LIN {X 0,Y 168.921,Z 1046.444,A -85,B 0,C 180,E1 28928.904,E2 28928.904} C_VEL
LIN {X 0,Y 193.808,Z 1028.505,A -85,B 0,C 180,E1 28941.439,E2 28941.439} C_VEL
LIN {X 0,Y 223.999,Z 1004.253,A -85,B 0,C 180,E1 28950.581,E2 28950.581} C_VEL
LIN {X 0,Y 255.108,Z 974.593,A -85,B 0,C 180,E1 28956.989,E2 28956.989} C_VEL
LIN {X 0,Y 284.282,Z 940.686,A -85,B 0,C 180,E1 28961.432,E2 28961.432} C_VEL
LIN {X 0,Y 287.15,Z 937.068,A -85,B 0,C 180,E1 28961.796,E2 28961.796} C_VEL
LIN {X 0,Y 289.842,Z 928.042,A -85,B 0,C 180,E1 28965.797,E2 28965.797} C_VEL
LIN {X 0,Y 291.827,Z 919.586,A -85,B 0,C 180,E1 28971.585,E2 28971.585} C_VEL
LIN {X 0,Y 293.357,Z 915.265,A -85,B 0,C 180,E1 28977.034,E2 28977.034} C_VEL
LIN {X 0,Y 293.788,Z 914.928,A -85,B 0,C 180,E1 28979.995,E2 28979.995} C_VEL
LIN {X 0,Y 292.859,Z 920.588,A -85,B 0,C 180,E1 28986.732,E2 28986.732} C_VEL
LIN {X 0,Y 291.654,Z 929.151,A -85,B 0,C 180,E1 28991.99,E2 28991.99} C_VEL
LIN {X 0,Y 290.091,Z 935.801,A -85,B 0,C 180,E1 28994.874,E2 28994.874} C_VEL
LIN {X 0,Y 261.778,Z 970.623,A -85,B 0,C 180,E1 28998.746,E2 28998.746} C_VEL
LIN {X 0,Y 232.501,Z 1000.468,A -85,B 0,C 180,E1 29004.144,E2 29004.144} C_VEL
LIN {X 0,Y 202.253,Z 1026.572,A -85,B 0,C 180,E1 29012.088,E2 29012.088} C_VEL
LIN {X 0,Y 173.882,Z 1048.21,A -85,B 0,C 180,E1 29024.19,E2 29024.19} C_VEL
LIN {X 0,Y 156.367,Z 1061.241,A -85,B 0,C 180,E1 29037.787,E2 29037.787} C_VEL
LIN {X 0,Y 148.038,Z 1068.795,A -85,B 0,C 180,E1 29052.113,E2 29052.113} C_VEL
LIN {X 0,Y 145.937,Z 1071.767,A -85,B 0,C 180,E1 29064.037,E2 29064.037} C_VEL
LIN {X 0,Y 146.316,Z 1072.302,A -85,B 0,C 180,E1 29069.997,E2 29069.997} C_VEL
LIN {X 0,Y 146.516,Z 1071.402,A -85,B 0,C 180,E1 29081.935,E2 29081.935} C_VEL
LIN {X 0,Y 151.978,Z 1066.921,A -85,B 0,C 180,E1 29096.206,E2 29096.206} C_VEL
LIN {X 0,Y 168.648,Z 1055.739,A -85,B 0,C 180,E1 29112.367,E2 29112.367} C_VEL
LIN {X 0,Y 194.431,Z 1038.433,A -85,B 0,C 180,E1 29124.918,E2 29124.918} C_VEL
LIN {X 0,Y 224.573,Z 1015.903,A -85,B 0,C 180,E1 29133.68,E2 29133.68} C_VEL
LIN {X 0,Y 256.304,Z 987.953,A -85,B 0,C 180,E1 29139.894,E2 29139.894} C_VEL
LIN {X 0,Y 288.623,Z 953.147,A -85,B 0,C 180,E1 29144.481,E2 29144.481} C_VEL
LIN {X 0,Y 296.037,Z 943.922,A -85,B 0,C 180,E1 29145.338,E2 29145.338} C_VEL
LIN {X 0,Y 297.368,Z 940.896,A -85,B 0,C 180,E1 29146.446,E2 29146.446} C_VEL
LIN {X 0,Y 299.07,Z 931.533,A -85,B 0,C 180,E1 29152.728,E2 29152.728} C_VEL
LIN {X 0,Y 299.728,Z 928.149,A -85,B 0,C 180,E1 29157.107,E2 29157.107} C_VEL
LIN {X 0,Y 299.819,Z 927.494,A -85,B 0,C 180,E1 29160.005,E2 29160.005} C_VEL
LIN {X 0,Y 297.474,Z 933.11,A -85,B 0,C 180,E1 29167.322,E2 29167.322} C_VEL
LIN {X 0,Y 294.947,Z 941.251,A -85,B 0,C 180,E1 29172.533,E2 29172.533} C_VEL
LIN {X 0,Y 293.335,Z 944.677,A -85,B 0,C 180,E1 29173.859,E2 29173.859} C_VEL
LIN {X 0,Y 263.75,Z 977.365,A -85,B 0,C 180,E1 29177.989,E2 29177.989} C_VEL
LIN {X 0,Y 233.929,Z 1004.507,A -85,B 0,C 180,E1 29183.498,E2 29183.498} C_VEL
LIN {X 0,Y 204.082,Z 1027.314,A -85,B 0,C 180,E1 29191.326,E2 29191.326} C_VEL
LIN {X 0,Y 176.268,Z 1045.628,A -85,B 0,C 180,E1 29202.828,E2 29202.828} C_VEL
LIN {X 0,Y 156.666,Z 1057.623,A -85,B 0,C 180,E1 29217.862,E2 29217.862} C_VEL
LIN {X 0,Y 148.093,Z 1063.059,A -85,B 0,C 180,E1 29232.125,E2 29232.125} C_VEL
LIN {X 0,Y 146.279,Z 1064.375,A -85,B 0,C 180,E1 29250.003,E2 29250.003} C_VEL
LIN {X 0,Y 147.555,Z 1062.344,A -85,B 0,C 180,E1 29261.856,E2 29261.856} C_VEL
LIN {X 0,Y 152.427,Z 1058.204,A -85,B 0,C 180,E1 29272.752,E2 29272.752} C_VEL
LIN {X 0,Y 153.265,Z 1055.117,A -85,B 0,C 180,E1 29279.211,E2 29279.211} C_VEL
LIN {X 0,Y 155.695,Z 1051.318,A -85,B 0,C 180,E1 29285.522,E2 29285.522} C_VEL
LIN {X 0,Y 179.336,Z 1035.523,A -85,B 0,C 180,E1 29299.512,E2 29299.512} C_VEL
LIN {X 0,Y 210.143,Z 1012.776,A -85,B 0,C 180,E1 29309.927,E2 29309.927} C_VEL
LIN {X 0,Y 242.764,Z 984.247,A -85,B 0,C 180,E1 29317.038,E2 29317.038} C_VEL
LIN {X 0,Y 274.308,Z 950.43,A -85,B 0,C 180,E1 29321.97,E2 29321.97} C_VEL
LIN {X 0,Y 282.718,Z 939.972,A -85,B 0,C 180,E1 29323.075,E2 29323.075} C_VEL
LIN {X 0,Y 285.788,Z 929.836,A -85,B 0,C 180,E1 29328.525,E2 29328.525} C_VEL
LIN {X 0,Y 287.675,Z 923.701,A -85,B 0,C 180,E1 29333.947,E2 29333.947} C_VEL
LIN {X 0,Y 288.554,Z 921.686,A -85,B 0,C 180,E1 29336.984,E2 29336.984} C_VEL
LIN {X 0,Y 289.013,Z 921.304,A -85,B 0,C 180,E1 29339.995,E2 29339.995} C_VEL
LIN {X 0,Y 288.103,Z 926.168,A -85,B 0,C 180,E1 29346.033,E2 29346.033} C_VEL
LIN {X 0,Y 286.388,Z 934.915,A -85,B 0,C 180,E1 29351.687,E2 29351.687} C_VEL
LIN {X 0,Y 285.234,Z 939.354,A -85,B 0,C 180,E1 29353.657,E2 29353.657} C_VEL
LIN {X 0,Y 254.602,Z 975.363,A -85,B 0,C 180,E1 29357.758,E2 29357.758} C_VEL
LIN {X 0,Y 222.094,Z 1006.526,A -85,B 0,C 180,E1 29363.799,E2 29363.799} C_VEL
LIN {X 0,Y 192.091,Z 1030.713,A -85,B 0,C 180,E1 29371.994,E2 29371.994} C_VEL
LIN {X 0,Y 166.418,Z 1049.188,A -85,B 0,C 180,E1 29383.238,E2 29383.238} C_VEL
LIN {X 0,Y 147.059,Z 1062.863,A -85,B 0,C 180,E1 29398.984,E2 29398.984} C_VEL
LIN {X 0,Y 140.394,Z 1068.559,A -85,B 0,C 180,E1 29411.103,E2 29411.103} C_VEL
LIN {X 0,Y 138.03,Z 1071.546,A -85,B 0,C 180,E1 29423.694,E2 29423.694} C_VEL
LIN {X 0,Y 138.396,Z 1072.088,A -85,B 0,C 180,E1 29429.997,E2 29429.997} C_VEL
LIN {X 0,Y 138.722,Z 1071.199,A -85,B 0,C 180,E1 29442.617,E2 29442.617} C_VEL
LIN {X 0,Y 144.75,Z 1066.727,A -85,B 0,C 180,E1 29457.623,E2 29457.623} C_VEL
LIN {X 0,Y 162.692,Z 1055.562,A -85,B 0,C 180,E1 29474.31,E2 29474.31} C_VEL
LIN {X 0,Y 189.855,Z 1038.279,A -85,B 0,C 180,E1 29486.936,E2 29486.936} C_VEL
LIN {X 0,Y 220.041,Z 1016.621,A -85,B 0,C 180,E1 29495.338,E2 29495.338} C_VEL
LIN {X 0,Y 253.534,Z 987.948,A -85,B 0,C 180,E1 29501.593,E2 29501.593} C_VEL
LIN {X 0,Y 286.881,Z 952.718,A -85,B 0,C 180,E1 29506.063,E2 29506.063} C_VEL
LIN {X 0,Y 291.416,Z 947.157,A -85,B 0,C 180,E1 29506.56,E2 29506.56} C_VEL
LIN {X 0,Y 293.48,Z 939.749,A -85,B 0,C 180,E1 29511.094,E2 29511.094} C_VEL
LIN {X 0,Y 294.665,Z 934.317,A -85,B 0,C 180,E1 29517.057,E2 29517.057} C_VEL
LIN {X 0,Y 294.769,Z 933.639,A -85,B 0,C 180,E1 29520.005,E2 29520.005} C_VEL
LIN {X 0,Y 292.789,Z 937.807,A -85,B 0,C 180,E1 29525.947,E2 29525.947} C_VEL
LIN {X 0,Y 289.965,Z 945.492,A -85,B 0,C 180,E1 29531.508,E2 29531.508} C_VEL
LIN {X 0,Y 288.508,Z 948.427,A -85,B 0,C 180,E1 29532.691,E2 29532.691} C_VEL
LIN {X 0,Y 256.762,Z 981.946,A -85,B 0,C 180,E1 29537.013,E2 29537.013} C_VEL
LIN {X 0,Y 224.354,Z 1009.714,A -85,B 0,C 180,E1 29543.035,E2 29543.035} C_VEL
LIN {X 0,Y 194.514,Z 1031.009,A -85,B 0,C 180,E1 29551.025,E2 29551.025} C_VEL
LIN {X 0,Y 168.277,Z 1047.332,A -85,B 0,C 180,E1 29562.219,E2 29562.219} C_VEL
LIN {X 0,Y 149.856,Z 1057.809,A -85,B 0,C 180,E1 29576.211,E2 29576.211} C_VEL
LIN {X 0,Y 140.48,Z 1063.256,A -85,B 0,C 180,E1 29591.121,E2 29591.121} C_VEL
LIN {X 0,Y 137.97,Z 1064.743,A -85,B 0,C 180,E1 29603.697,E2 29603.697} C_VEL
LIN {X 0,Y 138.358,Z 1064.59,A -85,B 0,C 180,E1 29610.003,E2 29610.003} C_VEL
LIN {X 0,Y 139.83,Z 1062.527,A -85,B 0,C 180,E1 29622.694,E2 29622.694} C_VEL
LIN {X 0,Y 150.114,Z 1055,A -85,B 0,C 180,E1 29640.318,E2 29640.318} C_VEL
LIN {X 0,Y 155.695,Z 1051.318,A -85,B 0,C 180,E1 29645.522,E2 29645.522} C_VEL
LIN {X 0,Y 159.585,Z 1046.926,A -85,B 0,C 180,E1 29651.527,E2 29651.527} C_VEL
LIN {X 0,Y 164.863,Z 1041.862,A -85,B 0,C 180,E1 29657.175,E2 29657.175} C_VEL
LIN {X 0,Y 194.943,Z 1021.511,A -85,B 0,C 180,E1 29668.774,E2 29668.774} C_VEL
LIN {X 0,Y 227.398,Z 995.695,A -85,B 0,C 180,E1 29676.562,E2 29676.562} C_VEL
LIN {X 0,Y 259.168,Z 965.038,A -85,B 0,C 180,E1 29681.84,E2 29681.84} C_VEL
LIN {X 0,Y 277.327,Z 944.261,A -85,B 0,C 180,E1 29684.24,E2 29684.24} C_VEL
LIN {X 0,Y 280.428,Z 936.455,A -85,B 0,C 180,E1 29688.34,E2 29688.34} C_VEL
LIN {X 0,Y 282.59,Z 930.048,A -85,B 0,C 180,E1 29693.838,E2 29693.838} C_VEL
LIN {X 0,Y 283.64,Z 928.013,A -85,B 0,C 180,E1 29696.932,E2 29696.932} C_VEL
LIN {X 0,Y 284.164,Z 927.612,A -85,B 0,C 180,E1 29699.994,E2 29699.994} C_VEL
LIN {X 0,Y 282.944,Z 932.529,A -85,B 0,C 180,E1 29706.143,E2 29706.143} C_VEL
LIN {X 0,Y 280.729,Z 942.17,A -85,B 0,C 180,E1 29712.183,E2 29712.183} C_VEL
LIN {X 0,Y 250.587,Z 976.786,A -85,B 0,C 180,E1 29716.25,E2 29716.25} C_VEL
LIN {X 0,Y 217.78,Z 1007.215,A -85,B 0,C 180,E1 29722.087,E2 29722.087} C_VEL
LIN {X 0,Y 185.18,Z 1032.411,A -85,B 0,C 180,E1 29730.763,E2 29730.763} C_VEL
LIN {X 0,Y 156.507,Z 1051.81,A -85,B 0,C 180,E1 29743.646,E2 29743.646} C_VEL
LIN {X 0,Y 137.865,Z 1064.196,A -85,B 0,C 180,E1 29760.264,E2 29760.264} C_VEL
LIN {X 0,Y 130.923,Z 1070.144,A -85,B 0,C 180,E1 29776.612,E2 29776.612} C_VEL
LIN {X 0,Y 130.474,Z 1071.873,A -85,B 0,C 180,E1 29789.997,E2 29789.997} C_VEL
LIN {X 0,Y 130.918,Z 1070.994,A -85,B 0,C 180,E1 29803.382,E2 29803.382} C_VEL
LIN {X 0,Y 138.027,Z 1066.297,A -85,B 0,C 180,E1 29819.77,E2 29819.77} C_VEL
LIN {X 0,Y 156.951,Z 1055.386,A -85,B 0,C 180,E1 29836.394,E2 29836.394} C_VEL
LIN {X 0,Y 185.533,Z 1038.125,A -85,B 0,C 180,E1 29849.046,E2 29849.046} C_VEL
LIN {X 0,Y 216.762,Z 1016.492,A -85,B 0,C 180,E1 29857.299,E2 29857.299} C_VEL
LIN {X 0,Y 251.084,Z 987.842,A -85,B 0,C 180,E1 29863.354,E2 29863.354} C_VEL
LIN {X 0,Y 285.551,Z 952.051,A -85,B 0,C 180,E1 29867.687,E2 29867.687} C_VEL
LIN {X 0,Y 286.562,Z 950.825,A -85,B 0,C 180,E1 29867.794,E2 29867.794} C_VEL
LIN {X 0,Y 288.661,Z 943.52,A -85,B 0,C 180,E1 29872.982,E2 29872.982} C_VEL
LIN {X 0,Y 289.525,Z 940.453,A -85,B 0,C 180,E1 29877.005,E2 29877.005} C_VEL
LIN {X 0,Y 289.661,Z 939.755,A -85,B 0,C 180,E1 29880.005,E2 29880.005} C_VEL
LIN {X 0,Y 287.31,Z 943.939,A -85,B 0,C 180,E1 29886.061,E2 29886.061} C_VEL
LIN {X 0,Y 284.553,Z 950.828,A -85,B 0,C 180,E1 29891.067,E2 29891.067} C_VEL
LIN {X 0,Y 282.419,Z 953.492,A -85,B 0,C 180,E1 29891.636,E2 29891.636} C_VEL
LIN {X 0,Y 251.817,Z 984.553,A -85,B 0,C 180,E1 29895.671,E2 29895.671} C_VEL
LIN {X 0,Y 218.2,Z 1012.227,A -85,B 0,C 180,E1 29901.742,E2 29901.742} C_VEL
LIN {X 0,Y 185.018,Z 1034.597,A -85,B 0,C 180,E1 29910.687,E2 29910.687} C_VEL
LIN {X 0,Y 156.681,Z 1050.874,A -85,B 0,C 180,E1 29923.69,E2 29923.69} C_VEL
LIN {X 0,Y 140.485,Z 1059.453,A -85,B 0,C 180,E1 29937.364,E2 29937.364} C_VEL
LIN {X 0,Y 130.891,Z 1064.502,A -85,B 0,C 180,E1 29956.615,E2 29956.615} C_VEL
LIN {X 0,Y 130.436,Z 1064.805,A -85,B 0,C 180,E1 29970.003,E2 29970.003} C_VEL
LIN {X 0,Y 132.06,Z 1062.801,A -85,B 0,C 180,E1 29983.271,E2 29983.271} C_VEL
LIN {X 0,Y 140.612,Z 1056.873,A -85,B 0,C 180,E1 29999.014,E2 29999.014} C_VEL
LIN {X 0,Y 159.276,Z 1045.31,A -85,B 0,C 180,E1 30014.143,E2 30014.143} C_VEL
LIN {X 0,Y 164.863,Z 1041.862,A -85,B 0,C 180,E1 30017.175,E2 30017.175} C_VEL
LIN {X 0,Y 171.332,Z 1036.252,A -85,B 0,C 180,E1 30022.395,E2 30022.395} C_VEL
LIN {X 0,Y 178.864,Z 1029.924,A -85,B 0,C 180,E1 30027.153,E2 30027.153} C_VEL
LIN {X 0,Y 211.654,Z 1006.358,A -85,B 0,C 180,E1 30035.91,E2 30035.91} C_VEL
LIN {X 0,Y 243.42,Z 978.764,A -85,B 0,C 180,E1 30041.63,E2 30041.63} C_VEL
LIN {X 0,Y 272.049,Z 948.544,A -85,B 0,C 180,E1 30045.463,E2 30045.463} C_VEL
LIN {X 0,Y 273.666,Z 945.717,A -85,B 0,C 180,E1 30046.464,E2 30046.464} C_VEL
LIN {X 0,Y 276.747,Z 938.05,A -85,B 0,C 180,E1 30051.968,E2 30051.968} C_VEL
LIN {X 0,Y 278.557,Z 934.205,A -85,B 0,C 180,E1 30056.876,E2 30056.876} C_VEL
LIN {X 0,Y 279.101,Z 933.771,A -85,B 0,C 180,E1 30059.994,E2 30059.994} C_VEL
LIN {X 0,Y 277.735,Z 938.902,A -85,B 0,C 180,E1 30066.259,E2 30066.259} C_VEL
LIN {X 0,Y 275.722,Z 945.879,A -85,B 0,C 180,E1 30070.88,E2 30070.88} C_VEL
LIN {X 0,Y 259.138,Z 965.305,A -85,B 0,C 180,E1 30073.043,E2 30073.043} C_VEL
LIN {X 0,Y 225.488,Z 997.948,A -85,B 0,C 180,E1 30078.082,E2 30078.082} C_VEL
LIN {X 0,Y 190.77,Z 1025.404,A -85,B 0,C 180,E1 30085.703,E2 30085.703} C_VEL
LIN {X 0,Y 157.942,Z 1047.279,A -85,B 0,C 180,E1 30097.665,E2 30097.665} C_VEL
LIN {X 0,Y 136.192,Z 1060.56,A -85,B 0,C 180,E1 30112.42,E2 30112.42} C_VEL
LIN {X 0,Y 125.26,Z 1068.086,A -85,B 0,C 180,E1 30128.716,E2 30128.716} C_VEL
LIN {X 0,Y 122.248,Z 1071.104,A -85,B 0,C 180,E1 30142.876,E2 30142.876} C_VEL
LIN {X 0,Y 122.551,Z 1071.658,A -85,B 0,C 180,E1 30149.997,E2 30149.997} C_VEL
LIN {X 0,Y 123.145,Z 1070.79,A -85,B 0,C 180,E1 30164.244,E2 30164.244} C_VEL
LIN {X 0,Y 130.946,Z 1066.16,A -85,B 0,C 180,E1 30181.38,E2 30181.38} C_VEL
LIN {X 0,Y 151.31,Z 1055.289,A -85,B 0,C 180,E1 30198.541,E2 30198.541} C_VEL
LIN {X 0,Y 181.469,Z 1037.972,A -85,B 0,C 180,E1 30211.257,E2 30211.257} C_VEL
LIN {X 0,Y 215.929,Z 1014.684,A -85,B 0,C 180,E1 30219.759,E2 30219.759} C_VEL
LIN {X 0,Y 250.58,Z 986.162,A -85,B 0,C 180,E1 30225.371,E2 30225.371} C_VEL
LIN {X 0,Y 281.749,Z 954.276,A -85,B 0,C 180,E1 30229.23,E2 30229.23} C_VEL
LIN {X 0,Y 283.743,Z 947.766,A -85,B 0,C 180,E1 30234.877,E2 30234.877} C_VEL
LIN {X 0,Y 284.331,Z 945.673,A -85,B 0,C 180,E1 30240.006,E2 30240.006} C_VEL
LIN {X 0,Y 281.804,Z 950.087,A -85,B 0,C 180,E1 30246.18,E2 30246.18} C_VEL
LIN {X 0,Y 279.498,Z 954.925,A -85,B 0,C 180,E1 30249.974,E2 30249.974} C_VEL
LIN {X 0,Y 247.647,Z 986.458,A -85,B 0,C 180,E1 30254.174,E2 30254.174} C_VEL
LIN {X 0,Y 213.74,Z 1013.469,A -85,B 0,C 180,E1 30260.052,E2 30260.052} C_VEL
LIN {X 0,Y 180.983,Z 1034.747,A -85,B 0,C 180,E1 30268.461,E2 30268.461} C_VEL
LIN {X 0,Y 150.83,Z 1051.214,A -85,B 0,C 180,E1 30281.632,E2 30281.632} C_VEL
LIN {X 0,Y 131.105,Z 1060.818,A -85,B 0,C 180,E1 30298.662,E2 30298.662} C_VEL
LIN {X 0,Y 123.137,Z 1064.706,A -85,B 0,C 180,E1 30315.755,E2 30315.755} C_VEL
LIN {X 0,Y 122.513,Z 1065.019,A -85,B 0,C 180,E1 30330.003,E2 30330.003} C_VEL
LIN {X 0,Y 124.361,Z 1063.029,A -85,B 0,C 180,E1 30344.109,E2 30344.109} C_VEL
LIN {X 0,Y 136.532,Z 1055.502,A -85,B 0,C 180,E1 30363.711,E2 30363.711} C_VEL
LIN {X 0,Y 159.702,Z 1042.017,A -85,B 0,C 180,E1 30379.39,E2 30379.39} C_VEL
LIN {X 0,Y 178.864,Z 1029.924,A -85,B 0,C 180,E1 30387.153,E2 30387.153} C_VEL
LIN {X 0,Y 187.324,Z 1023.081,A -85,B 0,C 180,E1 30391.469,E2 30391.469} C_VEL
LIN {X 0,Y 196.494,Z 1015.531,A -85,B 0,C 180,E1 30395.324,E2 30395.324} C_VEL
LIN {X 0,Y 229.476,Z 989.539,A -85,B 0,C 180,E1 30401.681,E2 30401.681} C_VEL
LIN {X 0,Y 261.489,Z 958.518,A -85,B 0,C 180,E1 30406.104,E2 30406.104} C_VEL
LIN {X 0,Y 268.247,Z 951.051,A -85,B 0,C 180,E1 30406.934,E2 30406.934} C_VEL
LIN {X 0,Y 271.279,Z 944.116,A -85,B 0,C 180,E1 30411.935,E2 30411.935} C_VEL
LIN {X 0,Y 273.381,Z 940.339,A -85,B 0,C 180,E1 30416.817,E2 30416.817} C_VEL
LIN {X 0,Y 273.99,Z 939.897,A -85,B 0,C 180,E1 30419.994,E2 30419.994} C_VEL
LIN {X 0,Y 272.261,Z 945.09,A -85,B 0,C 180,E1 30426.385,E2 30426.385} C_VEL
LIN {X 0,Y 270.711,Z 949.897,A -85,B 0,C 180,E1 30429.662,E2 30429.662} C_VEL
LIN {X 0,Y 239.67,Z 982.622,A -85,B 0,C 180,E1 30433.549,E2 30433.549} C_VEL
LIN {X 0,Y 208.084,Z 1009.77,A -85,B 0,C 180,E1 30438.777,E2 30438.777} C_VEL
LIN {X 0,Y 174.492,Z 1033.743,A -85,B 0,C 180,E1 30447.1,E2 30447.1} C_VEL
LIN {X 0,Y 144.446,Z 1052.051,A -85,B 0,C 180,E1 30459.717,E2 30459.717} C_VEL
LIN {X 0,Y 123.959,Z 1063.745,A -85,B 0,C 180,E1 30476.62,E2 30476.62} C_VEL
LIN {X 0,Y 115.394,Z 1069.686,A -85,B 0,C 180,E1 30494.769,E2 30494.769} C_VEL
LIN {X 0,Y 114.652,Z 1071.445,A -85,B 0,C 180,E1 30509.996,E2 30509.996} C_VEL
LIN {X 0,Y 115.392,Z 1070.585,A -85,B 0,C 180,E1 30525.224,E2 30525.224} C_VEL
LIN {X 0,Y 124.096,Z 1065.966,A -85,B 0,C 180,E1 30543.33,E2 30543.33} C_VEL
LIN {X 0,Y 145.076,Z 1055.606,A -85,B 0,C 180,E1 30560.413,E2 30560.413} C_VEL
LIN {X 0,Y 174.795,Z 1039.579,A -85,B 0,C 180,E1 30572.696,E2 30572.696} C_VEL
LIN {X 0,Y 210.303,Z 1016.735,A -85,B 0,C 180,E1 30581.259,E2 30581.259} C_VEL
LIN {X 0,Y 246.936,Z 987.628,A -85,B 0,C 180,E1 30586.954,E2 30586.954} C_VEL
LIN {X 0,Y 276.566,Z 958.292,A -85,B 0,C 180,E1 30590.49,E2 30590.49} C_VEL
LIN {X 0,Y 278.411,Z 953.302,A -85,B 0,C 180,E1 30595.323,E2 30595.323} C_VEL
LIN {X 0,Y 278.988,Z 951.574,A -85,B 0,C 180,E1 30600.006,E2 30600.006} C_VEL
LIN {X 0,Y 276.016,Z 956.022,A -85,B 0,C 180,E1 30606.31,E2 30606.31} C_VEL
LIN {X 0,Y 274.522,Z 958.994,A -85,B 0,C 180,E1 30608.765,E2 30608.765} C_VEL
LIN {X 0,Y 241.976,Z 989.783,A -85,B 0,C 180,E1 30612.859,E2 30612.859} C_VEL
LIN {X 0,Y 207.858,Z 1015.757,A -85,B 0,C 180,E1 30618.606,E2 30618.606} C_VEL
LIN {X 0,Y 174.361,Z 1036.519,A -85,B 0,C 180,E1 30627.026,E2 30627.026} C_VEL
LIN {X 0,Y 144.644,Z 1051.836,A -85,B 0,C 180,E1 30639.74,E2 30639.74} C_VEL
LIN {X 0,Y 124.258,Z 1061.011,A -85,B 0,C 180,E1 30656.719,E2 30656.719} C_VEL
LIN {X 0,Y 115.398,Z 1064.909,A -85,B 0,C 180,E1 30674.777,E2 30674.777} C_VEL
LIN {X 0,Y 114.617,Z 1065.233,A -85,B 0,C 180,E1 30690.004,E2 30690.004} C_VEL
LIN {X 0,Y 116.664,Z 1063.257,A -85,B 0,C 180,E1 30705.061,E2 30705.061} C_VEL
LIN {X 0,Y 129.94,Z 1055.753,A -85,B 0,C 180,E1 30725.674,E2 30725.674} C_VEL
LIN {X 0,Y 154.579,Z 1042.283,A -85,B 0,C 180,E1 30741.657,E2 30741.657} C_VEL
LIN {X 0,Y 188.739,Z 1021.037,A -85,B 0,C 180,E1 30753.401,E2 30753.401} C_VEL
LIN {X 0,Y 196.494,Z 1015.531,A -85,B 0,C 180,E1 30755.324,E2 30755.324} C_VEL
LIN {X 0,Y 206.235,Z 1007.478,A -85,B 0,C 180,E1 30758.786,E2 30758.786} C_VEL
LIN {X 0,Y 216.256,Z 998.768,A -85,B 0,C 180,E1 30761.897,E2 30761.897} C_VEL
LIN {X 0,Y 249.271,Z 969.538,A -85,B 0,C 180,E1 30766.586,E2 30766.586} C_VEL
LIN {X 0,Y 263.187,Z 955.082,A -85,B 0,C 180,E1 30768.2,E2 30768.2} C_VEL
LIN {X 0,Y 266.575,Z 948.64,A -85,B 0,C 180,E1 30773.466,E2 30773.466} C_VEL
LIN {X 0,Y 267.992,Z 946.329,A -85,B 0,C 180,E1 30776.753,E2 30776.753} C_VEL
LIN {X 0,Y 268.664,Z 945.808,A -85,B 0,C 180,E1 30779.994,E2 30779.994} C_VEL
LIN {X 0,Y 267.321,Z 949.42,A -85,B 0,C 180,E1 30784.872,E2 30784.872} C_VEL
LIN {X 0,Y 265.328,Z 954.401,A -85,B 0,C 180,E1 30788.522,E2 30788.522} C_VEL
LIN {X 0,Y 232.709,Z 987.152,A -85,B 0,C 180,E1 30792.359,E2 30792.359} C_VEL
LIN {X 0,Y 196.54,Z 1016.254,A -85,B 0,C 180,E1 30798.395,E2 30798.395} C_VEL
LIN {X 0,Y 160.778,Z 1039.637,A -85,B 0,C 180,E1 30807.86,E2 30807.86} C_VEL
LIN {X 0,Y 129.696,Z 1056.952,A -85,B 0,C 180,E1 30823.087,E2 30823.087} C_VEL
LIN {X 0,Y 110.411,Z 1067.612,A -85,B 0,C 180,E1 30845.681,E2 30845.681} C_VEL
LIN {X 0,Y 106.373,Z 1071.027,A -85,B 0,C 180,E1 30865.527,E2 30865.527} C_VEL
LIN {X 0,Y 106.4,Z 1071.286,A -85,B 0,C 180,E1 30874.653,E2 30874.653} C_VEL
LIN {X 0,Y 110.422,Z 1069.019,A -85,B 0,C 180,E1 30894.308,E2 30894.308} C_VEL
LIN {X 0,Y 127.838,Z 1061.135,A -85,B 0,C 180,E1 30915.332,E2 30915.332} C_VEL
LIN {X 0,Y 158.904,Z 1046.081,A -85,B 0,C 180,E1 30931.201,E2 30931.201} C_VEL
LIN {X 0,Y 195.775,Z 1024.678,A -85,B 0,C 180,E1 30941.07,E2 30941.07} C_VEL
LIN {X 0,Y 233.043,Z 997.752,A -85,B 0,C 180,E1 30947.257,E2 30947.257} C_VEL
LIN {X 0,Y 269.862,Z 964.234,A -85,B 0,C 180,E1 30951.432,E2 30951.432} C_VEL
LIN {X 0,Y 271.504,Z 962.226,A -85,B 0,C 180,E1 30951.934,E2 30951.934} C_VEL
LIN {X 0,Y 273.184,Z 958.02,A -85,B 0,C 180,E1 30956.826,E2 30956.826} C_VEL
LIN {X 0,Y 273.373,Z 957.268,A -85,B 0,C 180,E1 30960.006,E2 30960.006} C_VEL
LIN {X 0,Y 270.215,Z 961.942,A -85,B 0,C 180,E1 30966.446,E2 30966.446} C_VEL
LIN {X 0,Y 268.787,Z 963.916,A -85,B 0,C 180,E1 30967.702,E2 30967.702} C_VEL
LIN {X 0,Y 234.592,Z 994.666,A -85,B 0,C 180,E1 30971.766,E2 30971.766} C_VEL
LIN {X 0,Y 198.501,Z 1020.43,A -85,B 0,C 180,E1 30977.788,E2 30977.788} C_VEL
LIN {X 0,Y 163.083,Z 1040.716,A -85,B 0,C 180,E1 30987.072,E2 30987.072} C_VEL
LIN {X 0,Y 136.418,Z 1053.374,A -85,B 0,C 180,E1 30998.964,E2 30998.964} C_VEL
LIN {X 0,Y 114.865,Z 1062.375,A -85,B 0,C 180,E1 31018.153,E2 31018.153} C_VEL
LIN {X 0,Y 106.45,Z 1065.577,A -85,B 0,C 180,E1 31041.82,E2 31041.82} C_VEL
LIN {X 0,Y 106.691,Z 1065.448,A -85,B 0,C 180,E1 31050.004,E2 31050.004} C_VEL
LIN {X 0,Y 109.017,Z 1063.486,A -85,B 0,C 180,E1 31066.145,E2 31066.145} C_VEL
LIN {X 0,Y 123.508,Z 1056.004,A -85,B 0,C 180,E1 31087.846,E2 31087.846} C_VEL
LIN {X 0,Y 149.715,Z 1042.55,A -85,B 0,C 180,E1 31104.076,E2 31104.076} C_VEL
LIN {X 0,Y 183.612,Z 1022.378,A -85,B 0,C 180,E1 31115.216,E2 31115.216} C_VEL
LIN {X 0,Y 216.256,Z 998.768,A -85,B 0,C 180,E1 31121.897,E2 31121.897} C_VEL
LIN {X 0,Y 226.647,Z 989.528,A -85,B 0,C 180,E1 31124.667,E2 31124.667} C_VEL
LIN {X 0,Y 237.081,Z 979.659,A -85,B 0,C 180,E1 31127.151,E2 31127.151} C_VEL
LIN {X 0,Y 257.851,Z 959.524,A -85,B 0,C 180,E1 31129.513,E2 31129.513} C_VEL
LIN {X 0,Y 260.239,Z 955.708,A -85,B 0,C 180,E1 31132.184,E2 31132.184} C_VEL
LIN {X 0,Y 262.561,Z 952.255,A -85,B 0,C 180,E1 31136.685,E2 31136.685} C_VEL
LIN {X 0,Y 263.305,Z 951.73,A -85,B 0,C 180,E1 31139.994,E2 31139.994} C_VEL
LIN {X 0,Y 261.438,Z 955.979,A -85,B 0,C 180,E1 31145.529,E2 31145.529} C_VEL
LIN {X 0,Y 260.908,Z 957.296,A -85,B 0,C 180,E1 31146.665,E2 31146.665} C_VEL
LIN {X 0,Y 258.75,Z 959.957,A -85,B 0,C 180,E1 31147.327,E2 31147.327} C_VEL
LIN {X 0,Y 226.23,Z 990.94,A -85,B 0,C 180,E1 31151.009,E2 31151.009} C_VEL
LIN {X 0,Y 191.836,Z 1017.506,A -85,B 0,C 180,E1 31156.547,E2 31156.547} C_VEL
LIN {X 0,Y 155.476,Z 1040.282,A -85,B 0,C 180,E1 31165.75,E2 31165.75} C_VEL
LIN {X 0,Y 124.276,Z 1056.692,A -85,B 0,C 180,E1 31180.344,E2 31180.344} C_VEL
LIN {X 0,Y 103.111,Z 1067.375,A -85,B 0,C 180,E1 31203.834,E2 31203.834} C_VEL
LIN {X 0,Y 98.619,Z 1070.439,A -85,B 0,C 180,E1 31221.157,E2 31221.157} C_VEL
LIN {X 0,Y 98.807,Z 1071.016,A -85,B 0,C 180,E1 31229.996,E2 31229.996} C_VEL
LIN {X 0,Y 100.014,Z 1070.176,A -85,B 0,C 180,E1 31247.636,E2 31247.636} C_VEL
LIN {X 0,Y 114.309,Z 1064.216,A -85,B 0,C 180,E1 31271.513,E2 31271.513} C_VEL
LIN {X 0,Y 141.768,Z 1052.341,A -85,B 0,C 180,E1 31288.77,E2 31288.77} C_VEL
LIN {X 0,Y 177.68,Z 1033.833,A -85,B 0,C 180,E1 31300.063,E2 31300.063} C_VEL
LIN {X 0,Y 215.688,Z 1009.401,A -85,B 0,C 180,E1 31307.112,E2 31307.112} C_VEL
LIN {X 0,Y 251.29,Z 980.743,A -85,B 0,C 180,E1 31311.454,E2 31311.454} C_VEL
LIN {X 0,Y 266.158,Z 966.615,A -85,B 0,C 180,E1 31313.057,E2 31313.057} C_VEL
LIN {X 0,Y 267.543,Z 963.734,A -85,B 0,C 180,E1 31316.759,E2 31316.759} C_VEL
LIN {X 0,Y 267.758,Z 962.961,A -85,B 0,C 180,E1 31320.006,E2 31320.006} C_VEL
LIN {X 0,Y 264.434,Z 967.2,A -85,B 0,C 180,E1 31326.175,E2 31326.175} C_VEL
LIN {X 0,Y 230.877,Z 996.436,A -85,B 0,C 180,E1 31330.095,E2 31330.095} C_VEL
LIN {X 0,Y 193.008,Z 1022.51,A -85,B 0,C 180,E1 31336.113,E2 31336.113} C_VEL
LIN {X 0,Y 155.486,Z 1042.891,A -85,B 0,C 180,E1 31345.784,E2 31345.784} C_VEL
LIN {X 0,Y 126.735,Z 1055.438,A -85,B 0,C 180,E1 31358.999,E2 31358.999} C_VEL
LIN {X 0,Y 105.672,Z 1063.336,A -85,B 0,C 180,E1 31379.393,E2 31379.393} C_VEL
LIN {X 0,Y 98.574,Z 1065.786,A -85,B 0,C 180,E1 31401.161,E2 31401.161} C_VEL
LIN {X 0,Y 98.772,Z 1065.663,A -85,B 0,C 180,E1 31410.004,E2 31410.004} C_VEL
LIN {X 0,Y 101.4,Z 1063.714,A -85,B 0,C 180,E1 31427.395,E2 31427.395} C_VEL
LIN {X 0,Y 117.279,Z 1056.255,A -85,B 0,C 180,E1 31450.25,E2 31450.25} C_VEL
LIN {X 0,Y 145.145,Z 1042.816,A -85,B 0,C 180,E1 31466.647,E2 31466.647} C_VEL
LIN {X 0,Y 180.39,Z 1022.667,A -85,B 0,C 180,E1 31477.535,E2 31477.535} C_VEL
LIN {X 0,Y 216.712,Z 996.918,A -85,B 0,C 180,E1 31484.357,E2 31484.357} C_VEL
LIN {X 0,Y 237.081,Z 979.659,A -85,B 0,C 180,E1 31487.151,E2 31487.151} C_VEL
LIN {X 0,Y 243.507,Z 973.237,A -85,B 0,C 180,E1 31488.953,E2 31488.953} C_VEL
LIN {X 0,Y 250.028,Z 966.375,A -85,B 0,C 180,E1 31490.623,E2 31490.623} C_VEL
LIN {X 0,Y 253.944,Z 962.447,A -85,B 0,C 180,E1 31491.309,E2 31491.309} C_VEL
LIN {X 0,Y 256.874,Z 958.027,A -85,B 0,C 180,E1 31496.612,E2 31496.612} C_VEL
LIN {X 0,Y 257.626,Z 957.526,A -85,B 0,C 180,E1 31500.182,E2 31500.182} C_VEL
LIN {X 0,Y 255.624,Z 961.897,A -85,B 0,C 180,E1 31505.655,E2 31505.655} C_VEL
LIN {X 0,Y 221.396,Z 993.46,A -85,B 0,C 180,E1 31509.396,E2 31509.396} C_VEL
LIN {X 0,Y 186.15,Z 1019.5,A -85,B 0,C 180,E1 31514.817,E2 31514.817} C_VEL
LIN {X 0,Y 152.206,Z 1039.946,A -85,B 0,C 180,E1 31522.928,E2 31522.928} C_VEL
LIN {X 0,Y 119.153,Z 1056.431,A -85,B 0,C 180,E1 31537.351,E2 31537.351} C_VEL
LIN {X 0,Y 95.932,Z 1067.137,A -85,B 0,C 180,E1 31561.708,E2 31561.708} C_VEL
LIN {X 0,Y 90.748,Z 1070.217,A -85,B 0,C 180,E1 31580.383,E2 31580.383} C_VEL
LIN {X 0,Y 90.895,Z 1070.801,A -85,B 0,C 180,E1 31589.996,E2 31589.996} C_VEL
LIN {X 0,Y 92.394,Z 1069.971,A -85,B 0,C 180,E1 31609.145,E2 31609.145} C_VEL
LIN {X 0,Y 108.35,Z 1064.028,A -85,B 0,C 180,E1 31634.366,E2 31634.366} C_VEL
LIN {X 0,Y 137.704,Z 1052.165,A -85,B 0,C 180,E1 31651.682,E2 31651.682} C_VEL
LIN {X 0,Y 174.765,Z 1033.84,A -85,B 0,C 180,E1 31662.512,E2 31662.512} C_VEL
LIN {X 0,Y 212.267,Z 1010.487,A -85,B 0,C 180,E1 31668.991,E2 31668.991} C_VEL
LIN {X 0,Y 248.422,Z 982.234,A -85,B 0,C 180,E1 31673.114,E2 31673.114} C_VEL
LIN {X 0,Y 260.819,Z 970.811,A -85,B 0,C 180,E1 31674.454,E2 31674.454} C_VEL
LIN {X 0,Y 261.658,Z 969.203,A -85,B 0,C 180,E1 31676.686,E2 31676.686} C_VEL
LIN {X 0,Y 261.884,Z 968.43,A -85,B 0,C 180,E1 31680.006,E2 31680.006} C_VEL
LIN {X 0,Y 260.159,Z 970.285,A -85,B 0,C 180,E1 31683.345,E2 31683.345} C_VEL
LIN {X 0,Y 258.596,Z 972.16,A -85,B 0,C 180,E1 31685.005,E2 31685.005} C_VEL
LIN {X 0,Y 222.454,Z 1001.828,A -85,B 0,C 180,E1 31688.983,E2 31688.983} C_VEL
LIN {X 0,Y 187.69,Z 1024.481,A -85,B 0,C 180,E1 31694.342,E2 31694.342} C_VEL
LIN {X 0,Y 152.232,Z 1043.002,A -85,B 0,C 180,E1 31702.964,E2 31702.964} C_VEL
LIN {X 0,Y 121.767,Z 1055.618,A -85,B 0,C 180,E1 31716.015,E2 31716.015} C_VEL
LIN {X 0,Y 101.475,Z 1062.76,A -85,B 0,C 180,E1 31733.325,E2 31733.325} C_VEL
LIN {X 0,Y 90.724,Z 1065.995,A -85,B 0,C 180,E1 31760.389,E2 31760.389} C_VEL
LIN {X 0,Y 90.86,Z 1065.877,A -85,B 0,C 180,E1 31770.004,E2 31770.004} C_VEL
LIN {X 0,Y 93.839,Z 1063.943,A -85,B 0,C 180,E1 31788.848,E2 31788.848} C_VEL
LIN {X 0,Y 111.274,Z 1056.506,A -85,B 0,C 180,E1 31812.921,E2 31812.921} C_VEL
LIN {X 0,Y 140.877,Z 1043.082,A -85,B 0,C 180,E1 31829.384,E2 31829.384} C_VEL
LIN {X 0,Y 178.237,Z 1022.501,A -85,B 0,C 180,E1 31840.109,E2 31840.109} C_VEL
LIN {X 0,Y 216.138,Z 996.139,A -85,B 0,C 180,E1 31846.616,E2 31846.616} C_VEL
LIN {X 0,Y 250.028,Z 966.375,A -85,B 0,C 180,E1 31850.623,E2 31850.623} C_VEL
LIN {X 0,Y 252.137,Z 963.97,A -85,B 0,C 180,E1 31851.683,E2 31851.683} C_VEL
LIN {X 0,Y 250.851,Z 964.089,A -85,B 0,C 180,E1 31856.018,E2 31856.018} C_VEL
LIN {X 0,Y 252.091,Z 963.094,A -85,B 0,C 180,E1 31859.994,E2 31859.994} C_VEL
LIN {X 0,Y 250.633,Z 965.768,A -85,B 0,C 180,E1 31863.937,E2 31863.937} C_VEL
LIN {X 0,Y 248.694,Z 967.798,A -85,B 0,C 180,E1 31864.449,E2 31864.449} C_VEL
LIN {X 0,Y 214.248,Z 997.933,A -85,B 0,C 180,E1 31868.001,E2 31868.001} C_VEL
LIN {X 0,Y 175.633,Z 1024.696,A -85,B 0,C 180,E1 31873.901,E2 31873.901} C_VEL
LIN {X 0,Y 136.506,Z 1046.08,A -85,B 0,C 180,E1 31884.073,E2 31884.073} C_VEL
LIN {X 0,Y 102.548,Z 1061.142,A -85,B 0,C 180,E1 31902.359,E2 31902.359} C_VEL
LIN {X 0,Y 84.846,Z 1068.766,A -85,B 0,C 180,E1 31929.066,E2 31929.066} C_VEL
LIN {X 0,Y 82.964,Z 1070.586,A -85,B 0,C 180,E1 31949.995,E2 31949.995} C_VEL
LIN {X 0,Y 84.847,Z 1069.766,A -85,B 0,C 180,E1 31970.924,E2 31970.924} C_VEL
LIN {X 0,Y 102.693,Z 1063.84,A -85,B 0,C 180,E1 31997.541,E2 31997.541} C_VEL
LIN {X 0,Y 137.02,Z 1050.723,A -85,B 0,C 180,E1 32015.835,E2 32015.835} C_VEL
LIN {X 0,Y 175.872,Z 1031.912,A -85,B 0,C 180,E1 32025.769,E2 32025.769} C_VEL
LIN {X 0,Y 216.852,Z 1006.302,A -85,B 0,C 180,E1 32031.873,E2 32031.873} C_VEL
LIN {X 0,Y 253.758,Z 976.752,A -85,B 0,C 180,E1 32035.496,E2 32035.496} C_VEL
LIN {X 0,Y 255.538,Z 975.046,A -85,B 0,C 180,E1 32036.067,E2 32036.067} C_VEL
LIN {X 0,Y 255.99,Z 973.89,A -85,B 0,C 180,E1 32040.006,E2 32040.006} C_VEL
LIN {X 0,Y 253.907,Z 975.935,A -85,B 0,C 180,E1 32043.428,E2 32043.428} C_VEL
LIN {X 0,Y 215.916,Z 1005.809,A -85,B 0,C 180,E1 32047.552,E2 32047.552} C_VEL
LIN {X 0,Y 175.544,Z 1030.344,A -85,B 0,C 180,E1 32053.802,E2 32053.802} C_VEL
LIN {X 0,Y 136.567,Z 1048.542,A -85,B 0,C 180,E1 32064.126,E2 32064.126} C_VEL
LIN {X 0,Y 102.841,Z 1060.614,A -85,B 0,C 180,E1 32082.549,E2 32082.549} C_VEL
LIN {X 0,Y 84.919,Z 1065.724,A -85,B 0,C 180,E1 32109.095,E2 32109.095} C_VEL
LIN {X 0,Y 82.93,Z 1066.092,A -85,B 0,C 180,E1 32130.005,E2 32130.005} C_VEL
LIN {X 0,Y 86.346,Z 1064.172,A -85,B 0,C 180,E1 32150.554,E2 32150.554} C_VEL
LIN {X 0,Y 105.544,Z 1056.757,A -85,B 0,C 180,E1 32175.887,E2 32175.887} C_VEL
LIN {X 0,Y 139.488,Z 1042.16,A -85,B 0,C 180,E1 32193.178,E2 32193.178} C_VEL
LIN {X 0,Y 178.221,Z 1021.262,A -85,B 0,C 180,E1 32203.062,E2 32203.062} C_VEL
LIN {X 0,Y 216.193,Z 995.139,A -85,B 0,C 180,E1 32208.919,E2 32208.919} C_VEL
LIN {X 0,Y 248.794,Z 966.733,A -85,B 0,C 180,E1 32212.557,E2 32212.557} C_VEL
LIN {X 0,Y 250.851,Z 964.089,A -85,B 0,C 180,E1 32216.018,E2 32216.018} C_VEL
LIN {X 0,Y 249.811,Z 965.007,A -85,B 0,C 180,E1 32217.971,E2 32217.971} C_VEL
LIN {X 0,Y 245.805,Z 969.228,A -85,B 0,C 180,E1 32221.229,E2 32221.229} C_VEL
LIN {X 0,Y 245.264,Z 970.165,A -85,B 0,C 180,E1 32222.61,E2 32222.61} C_VEL
LIN {X 0,Y 210.612,Z 999.575,A -85,B 0,C 180,E1 32226.126,E2 32226.126} C_VEL
LIN {X 0,Y 173.853,Z 1024.404,A -85,B 0,C 180,E1 32231.289,E2 32231.289} C_VEL
LIN {X 0,Y 134.827,Z 1045.109,A -85,B 0,C 180,E1 32240.382,E2 32240.382} C_VEL
LIN {X 0,Y 98.073,Z 1060.594,A -85,B 0,C 180,E1 32258.154,E2 32258.154} C_VEL
LIN {X 0,Y 82.041,Z 1066.661,A -85,B 0,C 180,E1 32276.343,E2 32276.343} C_VEL
LIN {X 0,Y 75.072,Z 1069.772,A -85,B 0,C 180,E1 32298.349,E2 32298.349} C_VEL
LIN {X 0,Y 75.044,Z 1070.372,A -85,B 0,C 180,E1 32309.995,E2 32309.995} C_VEL
LIN {X 0,Y 77.404,Z 1069.561,A -85,B 0,C 180,E1 32333.046,E2 32333.046} C_VEL
LIN {X 0,Y 98.793,Z 1063.168,A -85,B 0,C 180,E1 32362.173,E2 32362.173} C_VEL
LIN {X 0,Y 133.314,Z 1050.798,A -85,B 0,C 180,E1 32378.853,E2 32378.853} C_VEL
LIN {X 0,Y 174.042,Z 1031.764,A -85,B 0,C 180,E1 32388.38,E2 32388.38} C_VEL
LIN {X 0,Y 215.235,Z 1006.605,A -85,B 0,C 180,E1 32393.94,E2 32393.94} C_VEL
LIN {X 0,Y 247.681,Z 981.459,A -85,B 0,C 180,E1 32396.893,E2 32396.893} C_VEL
LIN {X 0,Y 249.701,Z 979.624,A -85,B 0,C 180,E1 32397.452,E2 32397.452} C_VEL
LIN {X 0,Y 249.889,Z 979.125,A -85,B 0,C 180,E1 32400.006,E2 32400.006} C_VEL
LIN {X 0,Y 249.121,Z 979.763,A -85,B 0,C 180,E1 32401.291,E2 32401.291} C_VEL
LIN {X 0,Y 247.04,Z 981.583,A -85,B 0,C 180,E1 32402.255,E2 32402.255} C_VEL
LIN {X 0,Y 210.294,Z 1009.008,A -85,B 0,C 180,E1 32405.93,E2 32405.93} C_VEL
LIN {X 0,Y 173.678,Z 1030.542,A -85,B 0,C 180,E1 32411.196,E2 32411.196} C_VEL
LIN {X 0,Y 135.097,Z 1048.044,A -85,B 0,C 180,E1 32420.408,E2 32420.408} C_VEL
LIN {X 0,Y 99.38,Z 1060.229,A -85,B 0,C 180,E1 32437.605,E2 32437.605} C_VEL
LIN {X 0,Y 82.219,Z 1064.842,A -85,B 0,C 180,E1 32456.437,E2 32456.437} C_VEL
LIN {X 0,Y 75.071,Z 1066.414,A -85,B 0,C 180,E1 32478.36,E2 32478.36} C_VEL
LIN {X 0,Y 75.005,Z 1066.307,A -85,B 0,C 180,E1 32490.005,E2 32490.005} C_VEL
LIN {X 0,Y 78.942,Z 1064.401,A -85,B 0,C 180,E1 32512.583,E2 32512.583} C_VEL
LIN {X 0,Y 100.122,Z 1057.008,A -85,B 0,C 180,E1 32539.187,E2 32539.187} C_VEL
LIN {X 0,Y 135.766,Z 1042.569,A -85,B 0,C 180,E1 32556.113,E2 32556.113} C_VEL
LIN {X 0,Y 176.048,Z 1021.559,A -85,B 0,C 180,E1 32565.563,E2 32565.563} C_VEL
LIN {X 0,Y 216.312,Z 994.262,A -85,B 0,C 180,E1 32571.193,E2 32571.193} C_VEL
LIN {X 0,Y 243.779,Z 970.946,A -85,B 0,C 180,E1 32574.06,E2 32574.06} C_VEL
LIN {X 0,Y 245.203,Z 969.287,A -85,B 0,C 180,E1 32576.45,E2 32576.45} C_VEL
LIN {X 0,Y 246.242,Z 968.544,A -85,B 0,C 180,E1 32579.994,E2 32579.994} C_VEL
LIN {X 0,Y 245.805,Z 969.228,A -85,B 0,C 180,E1 32581.229,E2 32581.229} C_VEL
LIN {X 0,Y 242.806,Z 972.275,A -85,B 0,C 180,E1 32582.084,E2 32582.084} C_VEL
LIN {X 0,Y 228.336,Z 984.736,A -85,B 0,C 180,E1 32582.197,E2 32582.197} C_VEL
LIN {X 0,Y 188.688,Z 1014.037,A -85,B 0,C 180,E1 32586.331,E2 32586.331} C_VEL
LIN {X 0,Y 147.852,Z 1037.362,A -85,B 0,C 180,E1 32593.159,E2 32593.159} C_VEL
LIN {X 0,Y 107.846,Z 1054.937,A -85,B 0,C 180,E1 32605.916,E2 32605.916} C_VEL
LIN {X 0,Y 78.93,Z 1065.164,A -85,B 0,C 180,E1 32627.773,E2 32627.773} C_VEL
LIN {X 0,Y 67.267,Z 1069.55,A -85,B 0,C 180,E1 32656.974,E2 32656.974} C_VEL
LIN {X 0,Y 67.108,Z 1070.157,A -85,B 0,C 180,E1 32669.994,E2 32669.994} C_VEL
LIN {X 0,Y 70.073,Z 1069.356,A -85,B 0,C 180,E1 32695.621,E2 32695.621} C_VEL
LIN {X 0,Y 92.476,Z 1063.463,A -85,B 0,C 180,E1 32725.012,E2 32725.012} C_VEL
LIN {X 0,Y 127.9,Z 1051.64,A -85,B 0,C 180,E1 32741.407,E2 32741.407} C_VEL
LIN {X 0,Y 169.022,Z 1033.383,A -85,B 0,C 180,E1 32750.465,E2 32750.465} C_VEL
LIN {X 0,Y 208.988,Z 1010.107,A -85,B 0,C 180,E1 32755.559,E2 32755.559} C_VEL
LIN {X 0,Y 242.549,Z 985.489,A -85,B 0,C 180,E1 32758.414,E2 32758.414} C_VEL
LIN {X 0,Y 243.764,Z 984.305,A -85,B 0,C 180,E1 32760.006,E2 32760.006} C_VEL
LIN {X 0,Y 242.476,Z 985.372,A -85,B 0,C 180,E1 32760.724,E2 32760.724} C_VEL
LIN {X 0,Y 201.128,Z 1014.587,A -85,B 0,C 180,E1 32764.637,E2 32764.637} C_VEL
LIN {X 0,Y 157.908,Z 1037.613,A -85,B 0,C 180,E1 32771.076,E2 32771.076} C_VEL
LIN {X 0,Y 118.251,Z 1053.285,A -85,B 0,C 180,E1 32781.716,E2 32781.716} C_VEL
LIN {X 0,Y 83.266,Z 1063.339,A -85,B 0,C 180,E1 32803.29,E2 32803.29} C_VEL
LIN {X 0,Y 67.275,Z 1066.624,A -85,B 0,C 180,E1 32836.988,E2 32836.988} C_VEL
LIN {X 0,Y 67.072,Z 1066.522,A -85,B 0,C 180,E1 32850.006,E2 32850.006} C_VEL
LIN {X 0,Y 71.658,Z 1064.629,A -85,B 0,C 180,E1 32875.027,E2 32875.027} C_VEL
LIN {X 0,Y 95.074,Z 1057.259,A -85,B 0,C 180,E1 32902.847,E2 32902.847} C_VEL
LIN {X 0,Y 130.246,Z 1043.879,A -85,B 0,C 180,E1 32918.567,E2 32918.567} C_VEL
LIN {X 0,Y 170.706,Z 1023.821,A -85,B 0,C 180,E1 32927.564,E2 32927.564} C_VEL
LIN {X 0,Y 210.047,Z 998.388,A -85,B 0,C 180,E1 32932.764,E2 32932.764} C_VEL
LIN {X 0,Y 237.178,Z 976.627,A -85,B 0,C 180,E1 32935.294,E2 32935.294} C_VEL
LIN {X 0,Y 239.194,Z 974.832,A -85,B 0,C 180,E1 32936.361,E2 32936.361} C_VEL
LIN {X 0,Y 240.087,Z 974.414,A -85,B 0,C 180,E1 32940.831,E2 32940.831} C_VEL
LIN {X 0,Y 239.971,Z 974.606,A -85,B 0,C 180,E1 32941.179,E2 32941.179} C_VEL
LIN {X 0,Y 228.336,Z 984.736,A -85,B 0,C 180,E1 32942.197,E2 32942.197} C_VEL
LIN {X 0,Y 214.508,Z 995.521,A -85,B 0,C 180,E1 32942.364,E2 32942.364} C_VEL
LIN {X 0,Y 200.193,Z 1005.634,A -85,B 0,C 180,E1 32942.574,E2 32942.574} C_VEL
LIN {X 0,Y 156.956,Z 1031.726,A -85,B 0,C 180,E1 32948.097,E2 32948.097} C_VEL
LIN {X 0,Y 115.417,Z 1050.618,A -85,B 0,C 180,E1 32957.83,E2 32957.83} C_VEL
LIN {X 0,Y 77.608,Z 1063.64,A -85,B 0,C 180,E1 32978.635,E2 32978.635} C_VEL
LIN {X 0,Y 62.94,Z 1068.076,A -85,B 0,C 180,E1 33001.207,E2 33001.207} C_VEL
LIN {X 0,Y 59.17,Z 1069.942,A -85,B 0,C 180,E1 33029.993,E2 33029.993} C_VEL
LIN {X 0,Y 62.942,Z 1069.152,A -85,B 0,C 180,E1 33058.778,E2 33058.778} C_VEL
LIN {X 0,Y 88.054,Z 1063.275,A -85,B 0,C 180,E1 33089.363,E2 33089.363} C_VEL
LIN {X 0,Y 129.241,Z 1050.093,A -85,B 0,C 180,E1 33105.931,E2 33105.931} C_VEL
LIN {X 0,Y 171.507,Z 1031.467,A -85,B 0,C 180,E1 33113.713,E2 33113.713} C_VEL
LIN {X 0,Y 214.141,Z 1006.346,A -85,B 0,C 180,E1 33118.261,E2 33118.261} C_VEL
LIN {X 0,Y 231.414,Z 993.969,A -85,B 0,C 180,E1 33119.63,E2 33119.63} C_VEL
LIN {X 0,Y 191.623,Z 1019.929,A -85,B 0,C 180,E1 33123.267,E2 33123.267} C_VEL
LIN {X 0,Y 153.3,Z 1039.145,A -85,B 0,C 180,E1 33128.708,E2 33128.708} C_VEL
LIN {X 0,Y 112.241,Z 1054.46,A -85,B 0,C 180,E1 33139.086,E2 33139.086} C_VEL
LIN {X 0,Y 77.918,Z 1063.533,A -85,B 0,C 180,E1 33158.935,E2 33158.935} C_VEL
LIN {X 0,Y 59.537,Z 1066.833,A -85,B 0,C 180,E1 33195.261,E2 33195.261} C_VEL
LIN {X 0,Y 59.15,Z 1066.737,A -85,B 0,C 180,E1 33210.007,E2 33210.007} C_VEL
LIN {X 0,Y 64.531,Z 1064.858,A -85,B 0,C 180,E1 33238.019,E2 33238.019} C_VEL
LIN {X 0,Y 90.455,Z 1057.509,A -85,B 0,C 180,E1 33266.901,E2 33266.901} C_VEL
LIN {X 0,Y 127.521,Z 1044.145,A -85,B 0,C 180,E1 33281.94,E2 33281.94} C_VEL
LIN {X 0,Y 169.16,Z 1024.109,A -85,B 0,C 180,E1 33290.218,E2 33290.218} C_VEL
LIN {X 0,Y 209.189,Z 998.702,A -85,B 0,C 180,E1 33294.942,E2 33294.942} C_VEL
LIN {X 0,Y 233.349,Z 979.757,A -85,B 0,C 180,E1 33297.155,E2 33297.155} C_VEL
LIN {X 0,Y 234.11,Z 979.266,A -85,B 0,C 180,E1 33299.418,E2 33299.418} C_VEL
LIN {X 0,Y 226.665,Z 985.664,A -85,B 0,C 180,E1 33300.271,E2 33300.271} C_VEL
LIN {X 0,Y 200.193,Z 1005.634,A -85,B 0,C 180,E1 33302.574,E2 33302.574} C_VEL
LIN {X 0,Y 185.435,Z 1015.078,A -85,B 0,C 180,E1 33302.875,E2 33302.875} C_VEL
LIN {X 0,Y 170.254,Z 1023.782,A -85,B 0,C 180,E1 33303.261,E2 33303.261} C_VEL
LIN {X 0,Y 126.406,Z 1045.123,A -85,B 0,C 180,E1 33310.479,E2 33310.479} C_VEL
LIN {X 0,Y 84.103,Z 1060.155,A -85,B 0,C 180,E1 33325.71,E2 33325.71} C_VEL
LIN {X 0,Y 56.013,Z 1067.845,A -85,B 0,C 180,E1 33357.234,E2 33357.234} C_VEL
LIN {X 0,Y 51.228,Z 1069.727,A -85,B 0,C 180,E1 33389.992,E2 33389.992} C_VEL
LIN {X 0,Y 59.687,Z 1068.328,A -85,B 0,C 180,E1 33430.429,E2 33430.429} C_VEL
LIN {X 0,Y 90.294,Z 1061.473,A -85,B 0,C 180,E1 33457.366,E2 33457.366} C_VEL
LIN {X 0,Y 131.376,Z 1048.438,A -85,B 0,C 180,E1 33470.318,E2 33470.318} C_VEL
LIN {X 0,Y 174.527,Z 1029.369,A -85,B 0,C 180,E1 33476.852,E2 33476.852} C_VEL
LIN {X 0,Y 203.643,Z 1012.875,A -85,B 0,C 180,E1 33479.646,E2 33479.646} C_VEL
LIN {X 0,Y 163.305,Z 1034.387,A -85,B 0,C 180,E1 33484.044,E2 33484.044} C_VEL
LIN {X 0,Y 123.607,Z 1050.253,A -85,B 0,C 180,E1 33491.267,E2 33491.267} C_VEL
LIN {X 0,Y 84.311,Z 1061.381,A -85,B 0,C 180,E1 33506.024,E2 33506.024} C_VEL
LIN {X 0,Y 56.124,Z 1066.541,A -85,B 0,C 180,E1 33537.324,E2 33537.324} C_VEL
LIN {X 0,Y 51.211,Z 1066.952,A -85,B 0,C 180,E1 33570.008,E2 33570.008} C_VEL
LIN {X 0,Y 57.623,Z 1065.087,A -85,B 0,C 180,E1 33601.742,E2 33601.742} C_VEL
LIN {X 0,Y 86.334,Z 1057.76,A -85,B 0,C 180,E1 33631.368,E2 33631.368} C_VEL
LIN {X 0,Y 125.26,Z 1044.41,A -85,B 0,C 180,E1 33645.443,E2 33645.443} C_VEL
LIN {X 0,Y 167.98,Z 1024.397,A -85,B 0,C 180,E1 33652.923,E2 33652.923} C_VEL
LIN {X 0,Y 208.636,Z 999.016,A -85,B 0,C 180,E1 33657.129,E2 33657.129} C_VEL
LIN {X 0,Y 223.727,Z 987.734,A -85,B 0,C 180,E1 33658.288,E2 33658.288} C_VEL
LIN {X 0,Y 183.834,Z 1015.787,A -85,B 0,C 180,E1 33661.742,E2 33661.742} C_VEL
LIN {X 0,Y 170.254,Z 1023.782,A -85,B 0,C 180,E1 33663.261,E2 33663.261} C_VEL
LIN {X 0,Y 154.753,Z 1031.865,A -85,B 0,C 180,E1 33663.765,E2 33663.765} C_VEL
LIN {X 0,Y 138.839,Z 1039.014,A -85,B 0,C 180,E1 33664.426,E2 33664.426} C_VEL
LIN {X 0,Y 94.111,Z 1055.96,A -85,B 0,C 180,E1 33674.937,E2 33674.937} C_VEL
LIN {X 0,Y 57.916,Z 1065.705,A -85,B 0,C 180,E1 33698.272,E2 33698.272} C_VEL
LIN {X 0,Y 44.237,Z 1068.881,A -85,B 0,C 180,E1 33729.957,E2 33729.957} C_VEL
LIN {X 0,Y 43.292,Z 1069.512,A -85,B 0,C 180,E1 33749.991,E2 33749.991} C_VEL
LIN {X 0,Y 49.444,Z 1068.741,A -85,B 0,C 180,E1 33787.795,E2 33787.795} C_VEL
LIN {X 0,Y 80.97,Z 1062.899,A -85,B 0,C 180,E1 33819.34,E2 33819.34} C_VEL
LIN {X 0,Y 126.16,Z 1049.799,A -85,B 0,C 180,E1 33833.114,E2 33833.114} C_VEL
LIN {X 0,Y 170.31,Z 1031.252,A -85,B 0,C 180,E1 33839.141,E2 33839.141} C_VEL
LIN {X 0,Y 173.895,Z 1029.39,A -85,B 0,C 180,E1 33840.009,E2 33840.009} C_VEL
LIN {X 0,Y 130.274,Z 1047.684,A -85,B 0,C 180,E1 33845.924,E2 33845.924} C_VEL
LIN {X 0,Y 87.54,Z 1060.054,A -85,B 0,C 180,E1 33857.82,E2 33857.82} C_VEL
LIN {X 0,Y 58.111,Z 1065.639,A -85,B 0,C 180,E1 33878.537,E2 33878.537} C_VEL
LIN {X 0,Y 44.274,Z 1067.253,A -85,B 0,C 180,E1 33909.994,E2 33909.994} C_VEL
LIN {X 0,Y 43.285,Z 1067.166,A -85,B 0,C 180,E1 33930.009,E2 33930.009} C_VEL
LIN {X 0,Y 51.024,Z 1065.315,A -85,B 0,C 180,E1 33966.451,E2 33966.451} C_VEL
LIN {X 0,Y 82.788,Z 1058.01,A -85,B 0,C 180,E1 33996.251,E2 33996.251} C_VEL
LIN {X 0,Y 123.481,Z 1044.676,A -85,B 0,C 180,E1 34009.065,E2 34009.065} C_VEL
LIN {X 0,Y 167.182,Z 1024.684,A -85,B 0,C 180,E1 34015.652,E2 34015.652} C_VEL
LIN {X 0,Y 192.109,Z 1010.173,A -85,B 0,C 180,E1 34018.079,E2 34018.079} C_VEL
LIN {X 0,Y 185.67,Z 1014.332,A -85,B 0,C 180,E1 34019.018,E2 34019.018} C_VEL
LIN {X 0,Y 140.225,Z 1038.425,A -85,B 0,C 180,E1 34024.221,E2 34024.221} C_VEL
LIN {X 0,Y 138.839,Z 1039.014,A -85,B 0,C 180,E1 34024.426,E2 34024.426} C_VEL
LIN {X 0,Y 122.648,Z 1045.508,A -85,B 0,C 180,E1 34025.298,E2 34025.298} C_VEL
LIN {X 0,Y 106.256,Z 1051.217,A -85,B 0,C 180,E1 34026.484,E2 34026.484} C_VEL
LIN {X 0,Y 65.223,Z 1062.901,A -85,B 0,C 180,E1 34041.647,E2 34041.647} C_VEL
LIN {X 0,Y 43.35,Z 1067.383,A -85,B 0,C 180,E1 34065.628,E2 34065.628} C_VEL
LIN {X 0,Y 35.343,Z 1069.297,A -85,B 0,C 180,E1 34109.989,E2 34109.989} C_VEL
LIN {X 0,Y 45.408,Z 1068.275,A -85,B 0,C 180,E1 34158.176,E2 34158.176} C_VEL
LIN {X 0,Y 78.463,Z 1062.71,A -85,B 0,C 180,E1 34184.925,E2 34184.925} C_VEL
LIN {X 0,Y 125.442,Z 1049.631,A -85,B 0,C 180,E1 34196.829,E2 34196.829} C_VEL
LIN {X 0,Y 147.148,Z 1041.375,A -85,B 0,C 180,E1 34200.011,E2 34200.011} C_VEL
LIN {X 0,Y 106.767,Z 1055.004,A -85,B 0,C 180,E1 34206.547,E2 34206.547} C_VEL
LIN {X 0,Y 65.414,Z 1064.113,A -85,B 0,C 180,E1 34222.099,E2 34222.099} C_VEL
LIN {X 0,Y 36.866,Z 1067.463,A -85,B 0,C 180,E1 34265.74,E2 34265.74} C_VEL
LIN {X 0,Y 35.341,Z 1067.382,A -85,B 0,C 180,E1 34290.011,E2 34290.011} C_VEL
LIN {X 0,Y 44.866,Z 1065.544,A -85,B 0,C 180,E1 34332.507,E2 34332.507} C_VEL
LIN {X 0,Y 79.898,Z 1058.26,A -85,B 0,C 180,E1 34361.518,E2 34361.518} C_VEL
LIN {X 0,Y 125.501,Z 1043.731,A -85,B 0,C 180,E1 34373.305,E2 34373.305} C_VEL
LIN {X 0,Y 163.616,Z 1026.589,A -85,B 0,C 180,E1 34378.312,E2 34378.312} C_VEL
LIN {X 0,Y 121.469,Z 1045.693,A -85,B 0,C 180,E1 34383.526,E2 34383.526} C_VEL
LIN {X 0,Y 106.256,Z 1051.217,A -85,B 0,C 180,E1 34386.484,E2 34386.484} C_VEL
LIN {X 0,Y 89.623,Z 1056.154,A -85,B 0,C 180,E1 34388.072,E2 34388.072} C_VEL
LIN {X 0,Y 72.858,Z 1060.29,A -85,B 0,C 180,E1 34390.34,E2 34390.34} C_VEL
LIN {X 0,Y 38.01,Z 1067.151,A -85,B 0,C 180,E1 34417.102,E2 34417.102} C_VEL
LIN {X 0,Y 27.392,Z 1069.081,A -85,B 0,C 180,E1 34469.985,E2 34469.985} C_VEL
LIN {X 0,Y 38.009,Z 1068.33,A -85,B 0,C 180,E1 34522.863,E2 34522.863} C_VEL
LIN {X 0,Y 76.746,Z 1062.522,A -85,B 0,C 180,E1 34550.818,E2 34550.818} C_VEL
LIN {X 0,Y 119.845,Z 1051.185,A -85,B 0,C 180,E1 34560.013,E2 34560.013} C_VEL
LIN {X 0,Y 76.791,Z 1061.951,A -85,B 0,C 180,E1 34569.387,E2 34569.387} C_VEL
LIN {X 0,Y 38.126,Z 1067.155,A -85,B 0,C 180,E1 34597.368,E2 34597.368} C_VEL
LIN {X 0,Y 27.397,Z 1067.597,A -85,B 0,C 180,E1 34650.015,E2 34650.015} C_VEL
LIN {X 0,Y 39.368,Z 1065.773,A -85,B 0,C 180,E1 34700.357,E2 34700.357} C_VEL
LIN {X 0,Y 77.726,Z 1058.509,A -85,B 0,C 180,E1 34727.143,E2 34727.143} C_VEL
LIN {X 0,Y 124.281,Z 1044.211,A -85,B 0,C 180,E1 34736.908,E2 34736.908} C_VEL
LIN {X 0,Y 132.743,Z 1040.84,A -85,B 0,C 180,E1 34738.261,E2 34738.261} C_VEL
LIN {X 0,Y 91.275,Z 1055.451,A -85,B 0,C 180,E1 34744.974,E2 34744.974} C_VEL
LIN {X 0,Y 72.858,Z 1060.29,A -85,B 0,C 180,E1 34750.34,E2 34750.34} C_VEL
LIN {X 0,Y 56.07,Z 1063.611,A -85,B 0,C 180,E1 34753.795,E2 34753.795} C_VEL
LIN {X 0,Y 39.386,Z 1066.062,A -85,B 0,C 180,E1 34759.859,E2 34759.859} C_VEL
LIN {X 0,Y 19.438,Z 1068.866,A -85,B 0,C 180,E1 34829.979,E2 34829.979} C_VEL
LIN {X 0,Y 33.753,Z 1068.124,A -85,B 0,C 180,E1 34893.86,E2 34893.86} C_VEL
LIN {X 0,Y 75.873,Z 1062.334,A -85,B 0,C 180,E1 34916.91,E2 34916.91} C_VEL
LIN {X 0,Y 90.917,Z 1059.097,A -85,B 0,C 180,E1 34920.131,E2 34920.131} C_VEL
LIN {X 0,Y 46.995,Z 1066.237,A -85,B 0,C 180,E1 34934.71,E2 34934.71} C_VEL
LIN {X 0,Y 23.245,Z 1067.883,A -85,B 0,C 180,E1 34969.337,E2 34969.337} C_VEL
LIN {X 0,Y 19.448,Z 1067.812,A -85,B 0,C 180,E1 35010.021,E2 35010.021} C_VEL
LIN {X 0,Y 34.828,Z 1066.002,A -85,B 0,C 180,E1 35070.508,E2 35070.508} C_VEL
LIN {X 0,Y 76.345,Z 1058.756,A -85,B 0,C 180,E1 35093.008,E2 35093.008} C_VEL
LIN {X 0,Y 101.44,Z 1051.999,A -85,B 0,C 180,E1 35098.199,E2 35098.199} C_VEL
LIN {X 0,Y 61.119,Z 1062.407,A -85,B 0,C 180,E1 35107.303,E2 35107.303} C_VEL
LIN {X 0,Y 39.386,Z 1066.062,A -85,B 0,C 180,E1 35119.859,E2 35119.859} C_VEL
LIN {X 0,Y 27.464,Z 1067.5,A -85,B 0,C 180,E1 35129.196,E2 35129.196} C_VEL
LIN {X 0,Y 11.402,Z 1068.564,A -85,B 0,C 180,E1 35179.95,E2 35179.95} C_VEL
LIN {X 0,Y 31.053,Z 1067.918,A -85,B 0,C 180,E1 35267.368,E2 35267.368} C_VEL
LIN {X 0,Y 60.609,Z 1064.695,A -85,B 0,C 180,E1 35280.209,E2 35280.209} C_VEL
LIN {X 0,Y 17.965,Z 1068.093,A -85,B 0,C 180,E1 35312.526,E2 35312.526} C_VEL
LIN {X 0,Y 11.495,Z 1068.028,A -85,B 0,C 180,E1 35370.035,E2 35370.035} C_VEL
LIN {X 0,Y 31.673,Z 1066.23,A -85,B 0,C 180,E1 35443.159,E2 35443.159} C_VEL
LIN {X 0,Y 68.122,Z 1060.565,A -85,B 0,C 180,E1 35458.082,E2 35458.082} C_VEL
LIN {X 0,Y 31.062,Z 1066.688,A -85,B 0,C 180,E1 35472.59,E2 35472.59} C_VEL
LIN {X 0,Y 11.402,Z 1068.564,A -85,B 0,C 180,E1 35539.95,E2 35539.95} C_VEL
LIN {X 0,Y 10.655,Z 1068.718,A -85,B 0,C 180,E1 35585.686,E2 35585.686} C_VEL
LIN {X 0,Y 19.27,Z 1068.272,A -85,B 0,C 180,E1 35637.645,E2 35637.645} C_VEL
LIN {X 0,Y 23.704,Z 1068.148,A -85,B 0,C 180,E1 35640.066,E2 35640.066} C_VEL
LIN {X 0,Y 3.541,Z 1068.243,A -85,B 0,C 180,E1 35730.114,E2 35730.114} C_VEL
LIN {X 0,Y 29.523,Z 1066.554,A -85,B 0,C 180,E1 35817.831,E2 35817.831} C_VEL
LIN {X 0,Y 3.518,Z 1068.434,A -85,B 0,C 180,E1 35909.886,E2 35909.886} C_VEL
LIN {X 0,Y 19.27,Z 1068.272,A -85,B 0,C 180,E1 35997.645,E2 35997.645} C_VEL
LIN {X 0,Y 21.279,Z 1070.271,A -85,B 0,C 180,E1 35998.87,E2 35998.87} C_VEL
LIN {X 0,Y 21.279,Z 1088.5,A -85,B 0,C 180,E1 35998.87,E2 35998.87} C_VEL
LIN {X 0,Y 21.279,Z 1088.5,A -85,B 0,C 180,E1 35998.87,E2 35998.87}

QRS_NEXT_CUT()
PTP {E1 36177.319,E2 36177.319}
PTP {X 0,Y 759.843,A -85,B 0,C 180,E1 36177.319,E2 36177.319,E3 0,E4 0,E5 0,E6 0}
QRS_SPEED_INIT()
LIN {X 0,Y 759.843,Z 1088.5,A -85,B 0,C 180,E1 36177.319,E2 36177.319,E3 0,E4 0,E5 0,E6 0} C_VEL
LIN {X 0,Y 759.843,Z 336.65,A -85,B 0,C 180,E1 36177.319,E2 36177.319} C_VEL
LIN {X 0,Y 759.843,Z 328.572,A -85,B 0,C 180,E1 36177.319,E2 36177.319} C_VEL
LIN {X 0,Y 759.843,Z 326.572,A -85,B 0,C 180,E1 36177.169,E2 36177.169} C_VEL
LIN {X 0,Y 759.893,Z 326.569,A -85,B 0,C 180,E1 36174.564,E2 36174.564} C_VEL
LIN {X 0,Y 759.866,Z 326.575,A -85,B 0,C 180,E1 36171.601,E2 36171.601} C_VEL
LIN {X 0,Y 759.843,Z 326.572,A -85,B 0,C 180,E1 36169.077,E2 36169.077} C_VEL
LIN {X 0,Y 759.889,Z 326.569,A -85,B 0,C 180,E1 36166.454,E2 36166.454} C_VEL
LIN {X 0,Y 759.869,Z 326.575,A -85,B 0,C 180,E1 36163.487,E2 36163.487} C_VEL
LIN {X 0,Y 759.844,Z 326.572,A -85,B 0,C 180,E1 36160.953,E2 36160.953} C_VEL
LIN {X 0,Y 759.881,Z 326.569,A -85,B 0,C 180,E1 36158.381,E2 36158.381} C_VEL
LIN {X 0,Y 759.869,Z 326.575,A -85,B 0,C 180,E1 36155.346,E2 36155.346} C_VEL
LIN {X 0,Y 759.844,Z 326.572,A -85,B 0,C 180,E1 36152.818,E2 36152.818} C_VEL
LIN {X 0,Y 759.879,Z 326.569,A -85,B 0,C 180,E1 36150.259,E2 36150.259} C_VEL
LIN {X 0,Y 759.872,Z 326.575,A -85,B 0,C 180,E1 36147.229,E2 36147.229} C_VEL
LIN {X 0,Y 759.845,Z 326.572,A -85,B 0,C 180,E1 36144.673,E2 36144.673} C_VEL
LIN {X 0,Y 759.898,Z 326.568,A -85,B 0,C 180,E1 36141.989,E2 36141.989} C_VEL
LIN {X 0,Y 759.869,Z 326.575,A -85,B 0,C 180,E1 36139.052,E2 36139.052} C_VEL
LIN {X 0,Y 759.846,Z 326.571,A -85,B 0,C 180,E1 36136.51,E2 36136.51} C_VEL
LIN {X 0,Y 759.898,Z 326.568,A -85,B 0,C 180,E1 36133.857,E2 36133.857} C_VEL
LIN {X 0,Y 759.873,Z 326.576,A -85,B 0,C 180,E1 36130.942,E2 36130.942} C_VEL
LIN {X 0,Y 759.846,Z 326.573,A -85,B 0,C 180,E1 36128.397,E2 36128.397} C_VEL
LIN {X 0,Y 759.894,Z 326.569,A -85,B 0,C 180,E1 36125.748,E2 36125.748} C_VEL
LIN {X 0,Y 759.868,Z 326.579,A -85,B 0,C 180,E1 36122.77,E2 36122.77} C_VEL
LIN {X 0,Y 759.846,Z 326.656,A -85,B 0,C 180,E1 36122.25,E2 36122.25} C_VEL
LIN {X 0,Y 759.884,Z 347.643,A -85,B 0,C 180,E1 36120.755,E2 36120.755} C_VEL
LIN {X 0,Y 759.912,Z 584.911,A -85,B 0,C 180,E1 36118.177,E2 36118.177} C_VEL
LIN {X 0,Y 759.916,Z 736.017,A -85,B 0,C 180,E1 36116.55,E2 36116.55} C_VEL
LIN {X 0,Y 759.9,Z 759.461,A -85,B 0,C 180,E1 36116.182,E2 36116.182} C_VEL
LIN {X 0,Y 759.903,Z 781.523,A -85,B 0,C 180,E1 36115.701,E2 36115.701} C_VEL
LIN {X 0,Y 759.898,Z 801.218,A -85,B 0,C 180,E1 36115.172,E2 36115.172} C_VEL
LIN {X 0,Y 759.919,Z 824.386,A -85,B 0,C 180,E1 36114.421,E2 36114.421} C_VEL
LIN {X 0,Y 759.916,Z 844.946,A -85,B 0,C 180,E1 36113.619,E2 36113.619} C_VEL
LIN {X 0,Y 759.913,Z 864.955,A -85,B 0,C 180,E1 36112.724,E2 36112.724} C_VEL
LIN {X 0,Y 759.91,Z 887,A -85,B 0,C 180,E1 36111.578,E2 36111.578} C_VEL
LIN {X 0,Y 759.916,Z 905.657,A -85,B 0,C 180,E1 36110.471,E2 36110.471} C_VEL
LIN {X 0,Y 759.908,Z 925.564,A -85,B 0,C 180,E1 36109.125,E2 36109.125} C_VEL
LIN {X 0,Y 759.913,Z 942.712,A -85,B 0,C 180,E1 36107.814,E2 36107.814} C_VEL
LIN {X 0,Y 759.912,Z 959.488,A -85,B 0,C 180,E1 36106.355,E2 36106.355} C_VEL
LIN {X 0,Y 759.897,Z 973.888,A -85,B 0,C 180,E1 36104.946,E2 36104.946} C_VEL
LIN {X 0,Y 759.908,Z 988.501,A -85,B 0,C 180,E1 36103.313,E2 36103.313} C_VEL
LIN {X 0,Y 759.906,Z 1000.009,A -85,B 0,C 180,E1 36101.845,E2 36101.845} C_VEL
LIN {X 0,Y 759.912,Z 1012.038,A -85,B 0,C 180,E1 36100.079,E2 36100.079} C_VEL
LIN {X 0,Y 759.9,Z 1021.248,A -85,B 0,C 180,E1 36098.475,E2 36098.475} C_VEL
LIN {X 0,Y 759.894,Z 1029.42,A -85,B 0,C 180,E1 36096.801,E2 36096.801} C_VEL
LIN {X 0,Y 759.914,Z 1036.478,A -85,B 0,C 180,E1 36094.982,E2 36094.982} C_VEL
LIN {X 0,Y 759.893,Z 1041.296,A -85,B 0,C 180,E1 36093.395,E2 36093.395} C_VEL
LIN {X 0,Y 759.914,Z 1045.436,A -85,B 0,C 180,E1 36091.508,E2 36091.508} C_VEL
LIN {X 0,Y 759.902,Z 1047.622,A -85,B 0,C 180,E1 36089.774,E2 36089.774} C_VEL
LIN {X 0,Y 759.911,Z 1048.5,A -85,B 0,C 180,E1 36087.964,E2 36087.964} C_VEL
LIN {X 0,Y 759.903,Z 1047.636,A -85,B 0,C 180,E1 36086.152,E2 36086.152} C_VEL
LIN {X 0,Y 759.912,Z 1045.563,A -85,B 0,C 180,E1 36084.488,E2 36084.488} C_VEL
LIN {X 0,Y 759.895,Z 1041.501,A -85,B 0,C 180,E1 36082.591,E2 36082.591} C_VEL
LIN {X 0,Y 759.914,Z 1036.69,A -85,B 0,C 180,E1 36080.992,E2 36080.992} C_VEL
LIN {X 0,Y 759.893,Z 1029.632,A -85,B 0,C 180,E1 36079.154,E2 36079.154} C_VEL
LIN {X 0,Y 759.904,Z 1021.383,A -85,B 0,C 180,E1 36077.461,E2 36077.461} C_VEL
LIN {X 0,Y 759.912,Z 1012.276,A -85,B 0,C 180,E1 36075.871,E2 36075.871} C_VEL
LIN {X 0,Y 759.907,Z 1000.391,A -85,B 0,C 180,E1 36074.116,E2 36074.116} C_VEL
LIN {X 0,Y 759.908,Z 988.697,A -85,B 0,C 180,E1 36072.621,E2 36072.621} C_VEL
LIN {X 0,Y 759.903,Z 973.001,A -85,B 0,C 180,E1 36070.875,E2 36070.875} C_VEL
LIN {X 0,Y 759.909,Z 959.029,A -85,B 0,C 180,E1 36069.512,E2 36069.512} C_VEL
LIN {X 0,Y 759.915,Z 940.673,A -85,B 0,C 180,E1 36067.935,E2 36067.935} C_VEL
LIN {X 0,Y 759.917,Z 923.41,A -85,B 0,C 180,E1 36066.627,E2 36066.627} C_VEL
LIN {X 0,Y 759.914,Z 903.513,A -85,B 0,C 180,E1 36065.306,E2 36065.306} C_VEL
LIN {X 0,Y 759.91,Z 885.071,A -85,B 0,C 180,E1 36064.223,E2 36064.223} C_VEL
LIN {X 0,Y 759.915,Z 862.835,A -85,B 0,C 180,E1 36063.087,E2 36063.087} C_VEL
LIN {X 0,Y 759.918,Z 843.709,A -85,B 0,C 180,E1 36062.239,E2 36062.239} C_VEL
LIN {X 0,Y 759.913,Z 820.69,A -85,B 0,C 180,E1 36061.359,E2 36061.359} C_VEL
LIN {X 0,Y 759.903,Z 799.673,A -85,B 0,C 180,E1 36060.693,E2 36060.693} C_VEL
LIN {X 0,Y 759.9,Z 779.134,A -85,B 0,C 180,E1 36060.15,E2 36060.15} C_VEL
LIN {X 0,Y 759.908,Z 753.73,A -85,B 0,C 180,E1 36059.629,E2 36059.629} C_VEL
LIN {X 0,Y 759.917,Z 733.55,A -85,B 0,C 180,E1 36059.329,E2 36059.329} C_VEL
LIN {X 0,Y 759.917,Z 462.351,A -85,B 0,C 180,E1 36056.411,E2 36056.411} C_VEL
LIN {X 0,Y 759.883,Z 347.478,A -85,B 0,C 180,E1 36055.152,E2 36055.152} C_VEL
LIN {X 0,Y 759.844,Z 326.576,A -85,B 0,C 180,E1 36053.644,E2 36053.644} C_VEL
LIN {X 0,Y 759.867,Z 326.576,A -85,B 0,C 180,E1 36051.121,E2 36051.121} C_VEL
LIN {X 0,Y 759.892,Z 326.569,A -85,B 0,C 180,E1 36048.139,E2 36048.139} C_VEL
LIN {X 0,Y 759.844,Z 326.572,A -85,B 0,C 180,E1 36045.498,E2 36045.498} C_VEL
LIN {X 0,Y 759.868,Z 326.575,A -85,B 0,C 180,E1 36042.971,E2 36042.971} C_VEL
LIN {X 0,Y 759.884,Z 326.569,A -85,B 0,C 180,E1 36039.951,E2 36039.951} C_VEL
LIN {X 0,Y 759.843,Z 326.573,A -85,B 0,C 180,E1 36037.347,E2 36037.347} C_VEL
LIN {X 0,Y 759.87,Z 326.574,A -85,B 0,C 180,E1 36034.805,E2 36034.805} C_VEL
LIN {X 0,Y 759.877,Z 326.569,A -85,B 0,C 180,E1 36031.759,E2 36031.759} C_VEL
LIN {X 0,Y 759.843,Z 326.572,A -85,B 0,C 180,E1 36029.223,E2 36029.223} C_VEL
LIN {X 0,Y 759.868,Z 326.575,A -85,B 0,C 180,E1 36026.686,E2 36026.686} C_VEL
LIN {X 0,Y 759.882,Z 326.569,A -85,B 0,C 180,E1 36023.662,E2 36023.662} C_VEL
LIN {X 0,Y 759.842,Z 326.572,A -85,B 0,C 180,E1 36021.054,E2 36021.054} C_VEL
LIN {X 0,Y 759.865,Z 326.575,A -85,B 0,C 180,E1 36018.569,E2 36018.569} C_VEL
LIN {X 0,Y 759.888,Z 326.569,A -85,B 0,C 180,E1 36015.571,E2 36015.571} C_VEL
LIN {X 0,Y 759.843,Z 326.572,A -85,B 0,C 180,E1 36013.004,E2 36013.004} C_VEL
LIN {X 0,Y 759.855,Z 326.575,A -85,B 0,C 180,E1 36010.539,E2 36010.539} C_VEL
LIN {X 0,Y 759.916,Z 326.569,A -85,B 0,C 180,E1 36007.637,E2 36007.637} C_VEL
LIN {X 0,Y 759.844,Z 326.572,A -85,B 0,C 180,E1 36004.907,E2 36004.907} C_VEL
LIN {X 0,Y 759.854,Z 326.575,A -85,B 0,C 180,E1 36002.413,E2 36002.413} C_VEL
LIN {X 0,Y 759.918,Z 326.57,A -85,B 0,C 180,E1 35999.548,E2 35999.548} C_VEL
LIN {X 0,Y 759.846,Z 326.571,A -85,B 0,C 180,E1 35996.832,E2 35996.832} C_VEL
LIN {X 0,Y 759.849,Z 326.574,A -85,B 0,C 180,E1 35994.336,E2 35994.336} C_VEL
LIN {X 0,Y 759.916,Z 326.572,A -85,B 0,C 180,E1 35991.525,E2 35991.525} C_VEL
LIN {X 0,Y 759.849,Z 326.571,A -85,B 0,C 180,E1 35988.77,E2 35988.77} C_VEL
LIN {X 0,Y 759.844,Z 326.574,A -85,B 0,C 180,E1 35986.298,E2 35986.298} C_VEL
LIN {X 0,Y 759.915,Z 326.577,A -85,B 0,C 180,E1 35983.567,E2 35983.567} C_VEL
LIN {X 0,Y 759.853,Z 326.571,A -85,B 0,C 180,E1 35980.713,E2 35980.713} C_VEL
LIN {X 0,Y 759.84,Z 326.573,A -85,B 0,C 180,E1 35978.286,E2 35978.286} C_VEL
LIN {X 0,Y 759.872,Z 326.575,A -85,B 0,C 180,E1 35975.76,E2 35975.76} C_VEL
LIN {X 0,Y 759.872,Z 326.57,A -85,B 0,C 180,E1 35972.747,E2 35972.747} C_VEL
LIN {X 0,Y 759.84,Z 326.573,A -85,B 0,C 180,E1 35970.257,E2 35970.257} C_VEL
LIN {X 0,Y 759.854,Z 326.575,A -85,B 0,C 180,E1 35967.792,E2 35967.792} C_VEL
LIN {X 0,Y 759.91,Z 326.57,A -85,B 0,C 180,E1 35964.9,E2 35964.9} C_VEL
LIN {X 0,Y 759.845,Z 326.572,A -85,B 0,C 180,E1 35962.266,E2 35962.266} C_VEL
LIN {X 0,Y 759.842,Z 326.574,A -85,B 0,C 180,E1 35959.849,E2 35959.849} C_VEL
LIN {X 0,Y 759.909,Z 326.578,A -85,B 0,C 180,E1 35957.13,E2 35957.13} C_VEL
LIN {X 0,Y 759.855,Z 326.571,A -85,B 0,C 180,E1 35954.287,E2 35954.287} C_VEL
LIN {X 0,Y 759.839,Z 326.574,A -85,B 0,C 180,E1 35951.849,E2 35951.849} C_VEL
LIN {X 0,Y 759.877,Z 326.577,A -85,B 0,C 180,E1 35949.266,E2 35949.266} C_VEL
LIN {X 0,Y 759.863,Z 326.573,A -85,B 0,C 180,E1 35946.231,E2 35946.231} C_VEL
LIN {X 0,Y 759.857,Z 326.883,A -85,B 0,C 180,E1 35946.17,E2 35946.17} C_VEL
LIN {X 0,Y 759.903,Z 363.722,A -85,B 0,C 180,E1 35943.684,E2 35943.684} C_VEL
LIN {X 0,Y 759.914,Z 377.344,A -85,B 0,C 180,E1 35942.802,E2 35942.802} C_VEL
LIN {X 0,Y 759.918,Z 632.42,A -85,B 0,C 180,E1 35940.034,E2 35940.034} C_VEL
LIN {X 0,Y 759.915,Z 765.994,A -85,B 0,C 180,E1 35938.595,E2 35938.595} C_VEL
LIN {X 0,Y 759.897,Z 790.301,A -85,B 0,C 180,E1 35938.21,E2 35938.21} C_VEL
LIN {X 0,Y 759.902,Z 811.683,A -85,B 0,C 180,E1 35937.742,E2 35937.742} C_VEL
LIN {X 0,Y 759.901,Z 831.086,A -85,B 0,C 180,E1 35937.221,E2 35937.221} C_VEL
LIN {X 0,Y 759.919,Z 853.739,A -85,B 0,C 180,E1 35936.491,E2 35936.491} C_VEL
LIN {X 0,Y 759.916,Z 875.252,A -85,B 0,C 180,E1 35935.651,E2 35935.651} C_VEL
LIN {X 0,Y 759.913,Z 894.66,A -85,B 0,C 180,E1 35934.783,E2 35934.783} C_VEL
LIN {X 0,Y 759.911,Z 917.061,A -85,B 0,C 180,E1 35933.62,E2 35933.62} C_VEL
LIN {X 0,Y 759.907,Z 935.706,A -85,B 0,C 180,E1 35932.513,E2 35932.513} C_VEL
LIN {X 0,Y 759.909,Z 955.524,A -85,B 0,C 180,E1 35931.173,E2 35931.173} C_VEL
LIN {X 0,Y 759.917,Z 972.885,A -85,B 0,C 180,E1 35929.845,E2 35929.845} C_VEL
LIN {X 0,Y 759.909,Z 989.391,A -85,B 0,C 180,E1 35928.409,E2 35928.409} C_VEL
LIN {X 0,Y 759.903,Z 1003.947,A -85,B 0,C 180,E1 35926.984,E2 35926.984} C_VEL
LIN {X 0,Y 759.915,Z 1018.836,A -85,B 0,C 180,E1 35925.317,E2 35925.317} C_VEL
LIN {X 0,Y 759.898,Z 1030.589,A -85,B 0,C 180,E1 35923.812,E2 35923.812} C_VEL
LIN {X 0,Y 759.901,Z 1042.785,A -85,B 0,C 180,E1 35921.999,E2 35921.999} C_VEL
LIN {X 0,Y 759.91,Z 1051.555,A -85,B 0,C 180,E1 35920.462,E2 35920.462} C_VEL
LIN {X 0,Y 759.89,Z 1060.073,A -85,B 0,C 180,E1 35918.703,E2 35918.703} C_VEL
LIN {X 0,Y 759.919,Z 1066.726,A -85,B 0,C 180,E1 35916.953,E2 35916.953} C_VEL
LIN {X 0,Y 759.906,Z 1071.51,A -85,B 0,C 180,E1 35915.361,E2 35915.361} C_VEL
LIN {X 0,Y 759.917,Z 1075.671,A -85,B 0,C 180,E1 35913.395,E2 35913.395} C_VEL
LIN {X 0,Y 759.899,Z 1077.63,A -85,B 0,C 180,E1 35911.81,E2 35911.81} C_VEL
LIN {X 0,Y 759.92,Z 1078.5,A -85,B 0,C 180,E1 35910,E2 35910} C_VEL
LIN {X 0,Y 759.899,Z 1077.63,A -85,B 0,C 180,E1 35908.19,E2 35908.19} C_VEL
LIN {X 0,Y 759.918,Z 1075.559,A -85,B 0,C 180,E1 35906.53,E2 35906.53} C_VEL
LIN {X 0,Y 759.906,Z 1071.51,A -85,B 0,C 180,E1 35904.639,E2 35904.639} C_VEL
LIN {X 0,Y 759.919,Z 1066.726,A -85,B 0,C 180,E1 35903.047,E2 35903.047} C_VEL
LIN {X 0,Y 759.892,Z 1059.729,A -85,B 0,C 180,E1 35901.22,E2 35901.22} C_VEL
LIN {X 0,Y 759.91,Z 1051.555,A -85,B 0,C 180,E1 35899.538,E2 35899.538} C_VEL
LIN {X 0,Y 759.901,Z 1042.786,A -85,B 0,C 180,E1 35898.001,E2 35898.001} C_VEL
LIN {X 0,Y 759.898,Z 1030.589,A -85,B 0,C 180,E1 35896.188,E2 35896.188} C_VEL
LIN {X 0,Y 759.917,Z 1018.833,A -85,B 0,C 180,E1 35894.683,E2 35894.683} C_VEL
LIN {X 0,Y 759.903,Z 1003.948,A -85,B 0,C 180,E1 35893.016,E2 35893.016} C_VEL
LIN {X 0,Y 759.909,Z 989.391,A -85,B 0,C 180,E1 35891.591,E2 35891.591} C_VEL
LIN {X 0,Y 759.911,Z 971.366,A -85,B 0,C 180,E1 35890.035,E2 35890.035} C_VEL
LIN {X 0,Y 759.913,Z 954.42,A -85,B 0,C 180,E1 35888.746,E2 35888.746} C_VEL
LIN {X 0,Y 759.909,Z 934.383,A -85,B 0,C 180,E1 35887.405,E2 35887.405} C_VEL
LIN {X 0,Y 759.91,Z 915.991,A -85,B 0,C 180,E1 35886.32,E2 35886.32} C_VEL
LIN {X 0,Y 759.912,Z 893.9,A -85,B 0,C 180,E1 35885.182,E2 35885.182} C_VEL
LIN {X 0,Y 759.916,Z 874.865,A -85,B 0,C 180,E1 35884.332,E2 35884.332} C_VEL
LIN {X 0,Y 759.916,Z 852.82,A -85,B 0,C 180,E1 35883.475,E2 35883.475} C_VEL
LIN {X 0,Y 759.901,Z 831.087,A -85,B 0,C 180,E1 35882.779,E2 35882.779} C_VEL
LIN {X 0,Y 759.902,Z 811.685,A -85,B 0,C 180,E1 35882.258,E2 35882.258} C_VEL
LIN {X 0,Y 759.899,Z 789.26,A -85,B 0,C 180,E1 35881.768,E2 35881.768} C_VEL
LIN {X 0,Y 759.917,Z 765.997,A -85,B 0,C 180,E1 35881.405,E2 35881.405} C_VEL
LIN {X 0,Y 759.899,Z 499.217,A -85,B 0,C 180,E1 35878.53,E2 35878.53} C_VEL
LIN {X 0,Y 759.911,Z 376.685,A -85,B 0,C 180,E1 35877.173,E2 35877.173} C_VEL
LIN {X 0,Y 759.853,Z 337.913,A -85,B 0,C 180,E1 35874.582,E2 35874.582} C_VEL
LIN {X 0,Y 759.861,Z 326.575,A -85,B 0,C 180,E1 35873.784,E2 35873.784} C_VEL
LIN {X 0,Y 759.887,Z 326.577,A -85,B 0,C 180,E1 35870.808,E2 35870.808} C_VEL
LIN {X 0,Y 759.841,Z 326.574,A -85,B 0,C 180,E1 35868.252,E2 35868.252} C_VEL
LIN {X 0,Y 759.85,Z 326.572,A -85,B 0,C 180,E1 35865.779,E2 35865.779} C_VEL
LIN {X 0,Y 759.913,Z 326.575,A -85,B 0,C 180,E1 35862.968,E2 35862.968} C_VEL
LIN {X 0,Y 759.847,Z 326.574,A -85,B 0,C 180,E1 35860.249,E2 35860.249} C_VEL
LIN {X 0,Y 759.841,Z 326.572,A -85,B 0,C 180,E1 35857.823,E2 35857.823} C_VEL
LIN {X 0,Y 759.9,Z 326.569,A -85,B 0,C 180,E1 35855.193,E2 35855.193} C_VEL
LIN {X 0,Y 759.862,Z 326.575,A -85,B 0,C 180,E1 35852.293,E2 35852.293} C_VEL
LIN {X 0,Y 759.84,Z 326.573,A -85,B 0,C 180,E1 35849.83,E2 35849.83} C_VEL
LIN {X 0,Y 759.863,Z 326.57,A -85,B 0,C 180,E1 35847.338,E2 35847.338} C_VEL
LIN {X 0,Y 759.884,Z 326.576,A -85,B 0,C 180,E1 35844.322,E2 35844.322} C_VEL
LIN {X 0,Y 759.841,Z 326.574,A -85,B 0,C 180,E1 35841.783,E2 35841.783} C_VEL
LIN {X 0,Y 759.853,Z 326.571,A -85,B 0,C 180,E1 35839.287,E2 35839.287} C_VEL
LIN {X 0,Y 759.912,Z 326.577,A -85,B 0,C 180,E1 35836.355,E2 35836.355} C_VEL
LIN {X 0,Y 759.844,Z 326.574,A -85,B 0,C 180,E1 35833.702,E2 35833.702} C_VEL
LIN {X 0,Y 759.85,Z 326.571,A -85,B 0,C 180,E1 35831.23,E2 35831.23} C_VEL
LIN {X 0,Y 759.916,Z 326.573,A -85,B 0,C 180,E1 35828.398,E2 35828.398} C_VEL
LIN {X 0,Y 759.85,Z 326.574,A -85,B 0,C 180,E1 35825.664,E2 35825.664} C_VEL
LIN {X 0,Y 759.846,Z 326.571,A -85,B 0,C 180,E1 35823.168,E2 35823.168} C_VEL
LIN {X 0,Y 759.918,Z 326.569,A -85,B 0,C 180,E1 35820.452,E2 35820.452} C_VEL
LIN {X 0,Y 759.855,Z 326.575,A -85,B 0,C 180,E1 35817.587,E2 35817.587} C_VEL
LIN {X 0,Y 759.843,Z 326.572,A -85,B 0,C 180,E1 35817.169,E2 35817.169} C_VEL
LIN {X 0,Y 758.856,Z 326.699,A -85,B 0,C 180,E1 35816.588,E2 35816.588} C_VEL
LIN {X 0,Y 752.444,Z 327.495,A -85,B 0,C 180,E1 35814.962,E2 35814.962} C_VEL
LIN {X 0,Y 751.957,Z 327.557,A -85,B 0,C 180,E1 35814.539,E2 35814.539} C_VEL
LIN {X 0,Y 751.926,Z 327.564,A -85,B 0,C 180,E1 35811.589,E2 35811.589} C_VEL
LIN {X 0,Y 751.905,Z 327.56,A -85,B 0,C 180,E1 35809.038,E2 35809.038} C_VEL
LIN {X 0,Y 751.96,Z 327.558,A -85,B 0,C 180,E1 35806.387,E2 35806.387} C_VEL
LIN {X 0,Y 751.928,Z 327.564,A -85,B 0,C 180,E1 35803.467,E2 35803.467} C_VEL
LIN {X 0,Y 751.906,Z 327.561,A -85,B 0,C 180,E1 35800.905,E2 35800.905} C_VEL
LIN {X 0,Y 751.965,Z 327.556,A -85,B 0,C 180,E1 35798.223,E2 35798.223} C_VEL
LIN {X 0,Y 751.923,Z 327.563,A -85,B 0,C 180,E1 35795.263,E2 35795.263} C_VEL
LIN {X 0,Y 751.906,Z 327.561,A -85,B 0,C 180,E1 35792.777,E2 35792.777} C_VEL
LIN {X 0,Y 751.965,Z 327.556,A -85,B 0,C 180,E1 35790.09,E2 35790.09} C_VEL
LIN {X 0,Y 751.925,Z 327.563,A -85,B 0,C 180,E1 35787.143,E2 35787.143} C_VEL
LIN {X 0,Y 751.908,Z 327.561,A -85,B 0,C 180,E1 35784.604,E2 35784.604} C_VEL
LIN {X 0,Y 751.967,Z 327.558,A -85,B 0,C 180,E1 35781.904,E2 35781.904} C_VEL
LIN {X 0,Y 751.928,Z 327.565,A -85,B 0,C 180,E1 35779.036,E2 35779.036} C_VEL
LIN {X 0,Y 751.908,Z 327.559,A -85,B 0,C 180,E1 35776.461,E2 35776.461} C_VEL
LIN {X 0,Y 751.978,Z 327.557,A -85,B 0,C 180,E1 35773.744,E2 35773.744} C_VEL
LIN {X 0,Y 751.924,Z 327.564,A -85,B 0,C 180,E1 35770.83,E2 35770.83} C_VEL
LIN {X 0,Y 751.909,Z 327.562,A -85,B 0,C 180,E1 35768.293,E2 35768.293} C_VEL
LIN {X 0,Y 751.977,Z 327.56,A -85,B 0,C 180,E1 35765.526,E2 35765.526} C_VEL
LIN {X 0,Y 751.918,Z 327.57,A -85,B 0,C 180,E1 35762.631,E2 35762.631} C_VEL
LIN {X 0,Y 752.019,Z 328.205,A -85,B 0,C 180,E1 35762.544,E2 35762.544} C_VEL
LIN {X 0,Y 752.673,Z 330.551,A -85,B 0,C 180,E1 35762.339,E2 35762.339} C_VEL
LIN {X 0,Y 752.738,Z 347.819,A -85,B 0,C 180,E1 35761.104,E2 35761.104} C_VEL
LIN {X 0,Y 753.146,Z 351.266,A -85,B 0,C 180,E1 35761.045,E2 35761.045} C_VEL
LIN {X 0,Y 752.991,Z 587.579,A -85,B 0,C 180,E1 35758.455,E2 35758.455} C_VEL
LIN {X 0,Y 752.881,Z 736.326,A -85,B 0,C 180,E1 35756.838,E2 35756.838} C_VEL
LIN {X 0,Y 752.803,Z 761.088,A -85,B 0,C 180,E1 35756.439,E2 35756.439} C_VEL
LIN {X 0,Y 752.755,Z 782.475,A -85,B 0,C 180,E1 35755.964,E2 35755.964} C_VEL
LIN {X 0,Y 752.692,Z 803.068,A -85,B 0,C 180,E1 35755.401,E2 35755.401} C_VEL
LIN {X 0,Y 752.615,Z 827.719,A -85,B 0,C 180,E1 35754.572,E2 35754.572} C_VEL
LIN {X 0,Y 752.542,Z 847.477,A -85,B 0,C 180,E1 35753.782,E2 35753.782} C_VEL
LIN {X 0,Y 752.439,Z 869.885,A -85,B 0,C 180,E1 35752.745,E2 35752.745} C_VEL
LIN {X 0,Y 752.362,Z 889.573,A -85,B 0,C 180,E1 35751.682,E2 35751.682} C_VEL
LIN {X 0,Y 752.278,Z 909.967,A -85,B 0,C 180,E1 35750.437,E2 35750.437} C_VEL
LIN {X 0,Y 752.196,Z 928.613,A -85,B 0,C 180,E1 35749.127,E2 35749.127} C_VEL
LIN {X 0,Y 752.118,Z 947.271,A -85,B 0,C 180,E1 35747.644,E2 35747.644} C_VEL
LIN {X 0,Y 752.085,Z 962.369,A -85,B 0,C 180,E1 35746.281,E2 35746.281} C_VEL
LIN {X 0,Y 752.024,Z 979.192,A -85,B 0,C 180,E1 35744.554,E2 35744.554} C_VEL
LIN {X 0,Y 751.98,Z 991.869,A -85,B 0,C 180,E1 35743.064,E2 35743.064} C_VEL
LIN {X 0,Y 751.955,Z 1005.115,A -85,B 0,C 180,E1 35741.272,E2 35741.272} C_VEL
LIN {X 0,Y 751.932,Z 1014.93,A -85,B 0,C 180,E1 35739.723,E2 35739.723} C_VEL
LIN {X 0,Y 751.918,Z 1024.578,A -85,B 0,C 180,E1 35737.949,E2 35737.949} C_VEL
LIN {X 0,Y 751.919,Z 1032.319,A -85,B 0,C 180,E1 35736.183,E2 35736.183} C_VEL
LIN {X 0,Y 751.904,Z 1038.071,A -85,B 0,C 180,E1 35734.576,E2 35734.576} C_VEL
LIN {X 0,Y 751.913,Z 1043.37,A -85,B 0,C 180,E1 35732.591,E2 35732.591} C_VEL
LIN {X 0,Y 751.915,Z 1046.253,A -85,B 0,C 180,E1 35730.991,E2 35730.991} C_VEL
LIN {X 0,Y 751.913,Z 1048.154,A -85,B 0,C 180,E1 35729.162,E2 35729.162} C_VEL
LIN {X 0,Y 751.891,Z 1048.347,A -85,B 0,C 180,E1 35727.409,E2 35727.409} C_VEL
LIN {X 0,Y 751.918,Z 1047.283,A -85,B 0,C 180,E1 35725.729,E2 35725.729} C_VEL
LIN {X 0,Y 751.917,Z 1044.403,A -85,B 0,C 180,E1 35723.817,E2 35723.817} C_VEL
LIN {X 0,Y 751.915,Z 1040.55,A -85,B 0,C 180,E1 35722.18,E2 35722.18} C_VEL
LIN {X 0,Y 751.898,Z 1034.799,A -85,B 0,C 180,E1 35720.354,E2 35720.354} C_VEL
LIN {X 0,Y 751.919,Z 1027.386,A -85,B 0,C 180,E1 35718.572,E2 35718.572} C_VEL
LIN {X 0,Y 751.925,Z 1019.21,A -85,B 0,C 180,E1 35716.935,E2 35716.935} C_VEL
LIN {X 0,Y 751.938,Z 1008.38,A -85,B 0,C 180,E1 35715.129,E2 35715.129} C_VEL
LIN {X 0,Y 751.978,Z 997.883,A -85,B 0,C 180,E1 35713.627,E2 35713.627} C_VEL
LIN {X 0,Y 752.007,Z 984.331,A -85,B 0,C 180,E1 35711.932,E2 35711.932} C_VEL
LIN {X 0,Y 752.051,Z 970.413,A -85,B 0,C 180,E1 35710.425,E2 35710.425} C_VEL
LIN {X 0,Y 752.111,Z 954.372,A -85,B 0,C 180,E1 35708.883,E2 35708.883} C_VEL
LIN {X 0,Y 752.167,Z 937.802,A -85,B 0,C 180,E1 35707.49,E2 35707.49} C_VEL
LIN {X 0,Y 752.241,Z 918.335,A -85,B 0,C 180,E1 35706.041,E2 35706.041} C_VEL
LIN {X 0,Y 752.312,Z 900.432,A -85,B 0,C 180,E1 35704.872,E2 35704.872} C_VEL
LIN {X 0,Y 752.417,Z 879.19,A -85,B 0,C 180,E1 35703.65,E2 35703.65} C_VEL
LIN {X 0,Y 752.488,Z 859.592,A -85,B 0,C 180,E1 35702.671,E2 35702.671} C_VEL
LIN {X 0,Y 752.59,Z 838.022,A -85,B 0,C 180,E1 35701.729,E2 35701.729} C_VEL
LIN {X 0,Y 752.643,Z 815.482,A -85,B 0,C 180,E1 35700.907,E2 35700.907} C_VEL
LIN {X 0,Y 752.723,Z 795.82,A -85,B 0,C 180,E1 35700.299,E2 35700.299} C_VEL
LIN {X 0,Y 752.788,Z 770.26,A -85,B 0,C 180,E1 35699.661,E2 35699.661} C_VEL
LIN {X 0,Y 752.848,Z 750.065,A -85,B 0,C 180,E1 35699.278,E2 35699.278} C_VEL
LIN {X 0,Y 752.884,Z 728.753,A -85,B 0,C 180,E1 35698.976,E2 35698.976} C_VEL
LIN {X 0,Y 753.089,Z 467.381,A -85,B 0,C 180,E1 35696.147,E2 35696.147} C_VEL
LIN {X 0,Y 752.941,Z 348.669,A -85,B 0,C 180,E1 35694.825,E2 35694.825} C_VEL
LIN {X 0,Y 752.669,Z 347.331,A -85,B 0,C 180,E1 35694.786,E2 35694.786} C_VEL
LIN {X 0,Y 752.503,Z 329.753,A -85,B 0,C 180,E1 35693.504,E2 35693.504} C_VEL
LIN {X 0,Y 751.916,Z 327.57,A -85,B 0,C 180,E1 35693.309,E2 35693.309} C_VEL
LIN {X 0,Y 751.975,Z 327.561,A -85,B 0,C 180,E1 35690.438,E2 35690.438} C_VEL
LIN {X 0,Y 751.909,Z 327.561,A -85,B 0,C 180,E1 35687.678,E2 35687.678} C_VEL
LIN {X 0,Y 751.917,Z 327.564,A -85,B 0,C 180,E1 35685.136,E2 35685.136} C_VEL
LIN {X 0,Y 751.976,Z 327.559,A -85,B 0,C 180,E1 35682.285,E2 35682.285} C_VEL
LIN {X 0,Y 751.908,Z 327.56,A -85,B 0,C 180,E1 35679.531,E2 35679.531} C_VEL
LIN {X 0,Y 751.914,Z 327.563,A -85,B 0,C 180,E1 35677.042,E2 35677.042} C_VEL
LIN {X 0,Y 751.977,Z 327.56,A -85,B 0,C 180,E1 35674.202,E2 35674.202} C_VEL
LIN {X 0,Y 751.909,Z 327.56,A -85,B 0,C 180,E1 35671.419,E2 35671.419} C_VEL
LIN {X 0,Y 751.911,Z 327.563,A -85,B 0,C 180,E1 35668.95,E2 35668.95} C_VEL
LIN {X 0,Y 751.978,Z 327.562,A -85,B 0,C 180,E1 35666.164,E2 35666.164} C_VEL
LIN {X 0,Y 751.913,Z 327.56,A -85,B 0,C 180,E1 35663.346,E2 35663.346} C_VEL
LIN {X 0,Y 751.907,Z 327.562,A -85,B 0,C 180,E1 35660.879,E2 35660.879} C_VEL
LIN {X 0,Y 751.976,Z 327.565,A -85,B 0,C 180,E1 35658.128,E2 35658.128} C_VEL
LIN {X 0,Y 751.915,Z 327.56,A -85,B 0,C 180,E1 35655.266,E2 35655.266} C_VEL
LIN {X 0,Y 751.906,Z 327.562,A -85,B 0,C 180,E1 35652.753,E2 35652.753} C_VEL
LIN {X 0,Y 751.976,Z 327.564,A -85,B 0,C 180,E1 35649.954,E2 35649.954} C_VEL
LIN {X 0,Y 751.913,Z 327.56,A -85,B 0,C 180,E1 35647.104,E2 35647.104} C_VEL
LIN {X 0,Y 751.905,Z 327.562,A -85,B 0,C 180,E1 35644.653,E2 35644.653} C_VEL
LIN {X 0,Y 751.973,Z 327.566,A -85,B 0,C 180,E1 35641.905,E2 35641.905} C_VEL
LIN {X 0,Y 751.917,Z 327.56,A -85,B 0,C 180,E1 35639.009,E2 35639.009} C_VEL
LIN {X 0,Y 751.905,Z 327.562,A -85,B 0,C 180,E1 35636.493,E2 35636.493} C_VEL
LIN {X 0,Y 751.976,Z 327.565,A -85,B 0,C 180,E1 35633.74,E2 35633.74} C_VEL
LIN {X 0,Y 751.917,Z 327.56,A -85,B 0,C 180,E1 35630.895,E2 35630.895} C_VEL
LIN {X 0,Y 751.903,Z 327.561,A -85,B 0,C 180,E1 35628.416,E2 35628.416} C_VEL
LIN {X 0,Y 751.959,Z 327.566,A -85,B 0,C 180,E1 35625.759,E2 35625.759} C_VEL
LIN {X 0,Y 751.924,Z 327.56,A -85,B 0,C 180,E1 35622.83,E2 35622.83} C_VEL
LIN {X 0,Y 751.901,Z 327.561,A -85,B 0,C 180,E1 35620.307,E2 35620.307} C_VEL
LIN {X 0,Y 751.954,Z 327.566,A -85,B 0,C 180,E1 35617.648,E2 35617.648} C_VEL
LIN {X 0,Y 751.926,Z 327.56,A -85,B 0,C 180,E1 35614.722,E2 35614.722} C_VEL
LIN {X 0,Y 751.902,Z 327.562,A -85,B 0,C 180,E1 35612.169,E2 35612.169} C_VEL
LIN {X 0,Y 751.947,Z 327.565,A -85,B 0,C 180,E1 35609.56,E2 35609.56} C_VEL
LIN {X 0,Y 751.927,Z 327.56,A -85,B 0,C 180,E1 35606.597,E2 35606.597} C_VEL
LIN {X 0,Y 751.901,Z 327.562,A -85,B 0,C 180,E1 35604.082,E2 35604.082} C_VEL
LIN {X 0,Y 751.933,Z 327.565,A -85,B 0,C 180,E1 35601.513,E2 35601.513} C_VEL
LIN {X 0,Y 751.929,Z 327.56,A -85,B 0,C 180,E1 35598.474,E2 35598.474} C_VEL
LIN {X 0,Y 751.901,Z 327.563,A -85,B 0,C 180,E1 35595.898,E2 35595.898} C_VEL
LIN {X 0,Y 751.939,Z 327.566,A -85,B 0,C 180,E1 35593.326,E2 35593.326} C_VEL
LIN {X 0,Y 751.931,Z 327.561,A -85,B 0,C 180,E1 35590.36,E2 35590.36} C_VEL
LIN {X 0,Y 751.9,Z 327.564,A -85,B 0,C 180,E1 35587.81,E2 35587.81} C_VEL
LIN {X 0,Y 751.972,Z 327.565,A -85,B 0,C 180,E1 35586.563,E2 35586.563} C_VEL
LIN {X 0,Y 752.813,Z 331.086,A -85,B 0,C 180,E1 35586.271,E2 35586.271} C_VEL
LIN {X 0,Y 752.744,Z 367.134,A -85,B 0,C 180,E1 35583.819,E2 35583.819} C_VEL
LIN {X 0,Y 752.801,Z 377.401,A -85,B 0,C 180,E1 35583.151,E2 35583.151} C_VEL
LIN {X 0,Y 753.182,Z 380.848,A -85,B 0,C 180,E1 35583.093,E2 35583.093} C_VEL
LIN {X 0,Y 752.979,Z 638.162,A -85,B 0,C 180,E1 35580.278,E2 35580.278} C_VEL
LIN {X 0,Y 752.879,Z 766.53,A -85,B 0,C 180,E1 35578.881,E2 35578.881} C_VEL
LIN {X 0,Y 752.8,Z 791.576,A -85,B 0,C 180,E1 35578.474,E2 35578.474} C_VEL
LIN {X 0,Y 752.755,Z 812.708,A -85,B 0,C 180,E1 35578.003,E2 35578.003} C_VEL
LIN {X 0,Y 752.693,Z 833.682,A -85,B 0,C 180,E1 35577.428,E2 35577.428} C_VEL
LIN {X 0,Y 752.614,Z 857.11,A -85,B 0,C 180,E1 35576.64,E2 35576.64} C_VEL
LIN {X 0,Y 752.546,Z 876.248,A -85,B 0,C 180,E1 35575.879,E2 35575.879} C_VEL
LIN {X 0,Y 752.469,Z 897.462,A -85,B 0,C 180,E1 35574.912,E2 35574.912} C_VEL
LIN {X 0,Y 752.363,Z 918.518,A -85,B 0,C 180,E1 35573.788,E2 35573.788} C_VEL
LIN {X 0,Y 752.292,Z 938.354,A -85,B 0,C 180,E1 35572.589,E2 35572.589} C_VEL
LIN {X 0,Y 752.2,Z 957.679,A -85,B 0,C 180,E1 35571.241,E2 35571.241} C_VEL
LIN {X 0,Y 752.131,Z 975.816,A -85,B 0,C 180,E1 35569.816,E2 35569.816} C_VEL
LIN {X 0,Y 752.084,Z 991.944,A -85,B 0,C 180,E1 35568.366,E2 35568.366} C_VEL
LIN {X 0,Y 752.018,Z 1007.676,A -85,B 0,C 180,E1 35566.77,E2 35566.77} C_VEL
LIN {X 0,Y 751.997,Z 1020.607,A -85,B 0,C 180,E1 35565.264,E2 35565.264} C_VEL
LIN {X 0,Y 751.967,Z 1033.325,A -85,B 0,C 180,E1 35563.587,E2 35563.587} C_VEL
LIN {X 0,Y 751.924,Z 1044.175,A -85,B 0,C 180,E1 35561.895,E2 35561.895} C_VEL
LIN {X 0,Y 751.931,Z 1052.78,A -85,B 0,C 180,E1 35560.342,E2 35560.342} C_VEL
LIN {X 0,Y 751.904,Z 1061.598,A -85,B 0,C 180,E1 35558.411,E2 35558.411} C_VEL
LIN {X 0,Y 751.906,Z 1067.489,A -85,B 0,C 180,E1 35556.797,E2 35556.797} C_VEL
LIN {X 0,Y 751.916,Z 1072.701,A -85,B 0,C 180,E1 35554.959,E2 35554.959} C_VEL
LIN {X 0,Y 751.916,Z 1076.121,A -85,B 0,C 180,E1 35553.125,E2 35553.125} C_VEL
LIN {X 0,Y 751.903,Z 1078.099,A -85,B 0,C 180,E1 35551.295,E2 35551.295} C_VEL
LIN {X 0,Y 751.891,Z 1078.351,A -85,B 0,C 180,E1 35549.467,E2 35549.467} C_VEL
LIN {X 0,Y 751.913,Z 1077.296,A -85,B 0,C 180,E1 35547.79,E2 35547.79} C_VEL
LIN {X 0,Y 751.91,Z 1074.343,A -85,B 0,C 180,E1 35545.832,E2 35545.832} C_VEL
LIN {X 0,Y 751.916,Z 1070.687,A -85,B 0,C 180,E1 35544.276,E2 35544.276} C_VEL
LIN {X 0,Y 751.897,Z 1064.936,A -85,B 0,C 180,E1 35542.435,E2 35542.435} C_VEL
LIN {X 0,Y 751.919,Z 1057.524,A -85,B 0,C 180,E1 35540.647,E2 35540.647} C_VEL
LIN {X 0,Y 751.924,Z 1049.516,A -85,B 0,C 180,E1 35539.038,E2 35539.038} C_VEL
LIN {X 0,Y 751.948,Z 1038.35,A -85,B 0,C 180,E1 35537.17,E2 35537.17} C_VEL
LIN {X 0,Y 751.97,Z 1027.951,A -85,B 0,C 180,E1 35535.681,E2 35535.681} C_VEL
LIN {X 0,Y 751.999,Z 1014.677,A -85,B 0,C 180,E1 35534.016,E2 35534.016} C_VEL
LIN {X 0,Y 752.053,Z 1000.842,A -85,B 0,C 180,E1 35532.514,E2 35532.514} C_VEL
LIN {X 0,Y 752.108,Z 984.651,A -85,B 0,C 180,E1 35530.952,E2 35530.952} C_VEL
LIN {X 0,Y 752.165,Z 967.82,A -85,B 0,C 180,E1 35529.536,E2 35529.536} C_VEL
LIN {X 0,Y 752.242,Z 948.443,A -85,B 0,C 180,E1 35528.094,E2 35528.094} C_VEL
LIN {X 0,Y 752.311,Z 930.417,A -85,B 0,C 180,E1 35526.916,E2 35526.916} C_VEL
LIN {X 0,Y 752.415,Z 908.748,A -85,B 0,C 180,E1 35525.672,E2 35525.672} C_VEL
LIN {X 0,Y 752.488,Z 889.454,A -85,B 0,C 180,E1 35524.71,E2 35524.71} C_VEL
LIN {X 0,Y 752.594,Z 867.166,A -85,B 0,C 180,E1 35523.741,E2 35523.741} C_VEL
LIN {X 0,Y 752.646,Z 846.235,A -85,B 0,C 180,E1 35522.977,E2 35522.977} C_VEL
LIN {X 0,Y 752.717,Z 827.025,A -85,B 0,C 180,E1 35522.379,E2 35522.379} C_VEL
LIN {X 0,Y 752.782,Z 802.762,A -85,B 0,C 180,E1 35521.758,E2 35521.758} C_VEL
LIN {X 0,Y 752.842,Z 781.048,A -85,B 0,C 180,E1 35521.339,E2 35521.339} C_VEL
LIN {X 0,Y 752.883,Z 760.645,A -85,B 0,C 180,E1 35521.045,E2 35521.045} C_VEL
LIN {X 0,Y 753.066,Z 501.507,A -85,B 0,C 180,E1 35518.236,E2 35518.236} C_VEL
LIN {X 0,Y 753.009,Z 378.268,A -85,B 0,C 180,E1 35516.869,E2 35516.869} C_VEL
LIN {X 0,Y 752.714,Z 376.593,A -85,B 0,C 180,E1 35516.812,E2 35516.812} C_VEL
LIN {X 0,Y 752.785,Z 339.845,A -85,B 0,C 180,E1 35514.331,E2 35514.331} C_VEL
LIN {X 0,Y 752.791,Z 330.294,A -85,B 0,C 180,E1 35513.673,E2 35513.673} C_VEL
LIN {X 0,Y 751.973,Z 327.564,A -85,B 0,C 180,E1 35513.431,E2 35513.431} C_VEL
LIN {X 0,Y 751.916,Z 327.567,A -85,B 0,C 180,E1 35510.533,E2 35510.533} C_VEL
LIN {X 0,Y 751.902,Z 327.563,A -85,B 0,C 180,E1 35508.018,E2 35508.018} C_VEL
LIN {X 0,Y 751.97,Z 327.559,A -85,B 0,C 180,E1 35505.299,E2 35505.299} C_VEL
LIN {X 0,Y 751.917,Z 327.564,A -85,B 0,C 180,E1 35502.393,E2 35502.393} C_VEL
LIN {X 0,Y 751.902,Z 327.561,A -85,B 0,C 180,E1 35499.888,E2 35499.888} C_VEL
LIN {X 0,Y 751.965,Z 327.558,A -85,B 0,C 180,E1 35497.204,E2 35497.204} C_VEL
LIN {X 0,Y 751.923,Z 327.564,A -85,B 0,C 180,E1 35494.321,E2 35494.321} C_VEL
LIN {X 0,Y 751.901,Z 327.562,A -85,B 0,C 180,E1 35491.777,E2 35491.777} C_VEL
LIN {X 0,Y 751.942,Z 327.559,A -85,B 0,C 180,E1 35489.21,E2 35489.21} C_VEL
LIN {X 0,Y 751.926,Z 327.564,A -85,B 0,C 180,E1 35486.199,E2 35486.199} C_VEL
LIN {X 0,Y 751.902,Z 327.561,A -85,B 0,C 180,E1 35483.679,E2 35483.679} C_VEL
LIN {X 0,Y 751.937,Z 327.559,A -85,B 0,C 180,E1 35481.123,E2 35481.123} C_VEL
LIN {X 0,Y 751.934,Z 327.565,A -85,B 0,C 180,E1 35478.129,E2 35478.129} C_VEL
LIN {X 0,Y 751.903,Z 327.562,A -85,B 0,C 180,E1 35475.582,E2 35475.582} C_VEL
LIN {X 0,Y 751.937,Z 327.558,A -85,B 0,C 180,E1 35472.987,E2 35472.987} C_VEL
LIN {X 0,Y 751.93,Z 327.563,A -85,B 0,C 180,E1 35469.955,E2 35469.955} C_VEL
LIN {X 0,Y 751.903,Z 327.562,A -85,B 0,C 180,E1 35467.411,E2 35467.411} C_VEL
LIN {X 0,Y 751.943,Z 327.558,A -85,B 0,C 180,E1 35464.806,E2 35464.806} C_VEL
LIN {X 0,Y 751.932,Z 327.565,A -85,B 0,C 180,E1 35461.829,E2 35461.829} C_VEL
LIN {X 0,Y 751.905,Z 327.56,A -85,B 0,C 180,E1 35459.314,E2 35459.314} C_VEL
LIN {X 0,Y 751.937,Z 327.559,A -85,B 0,C 180,E1 35456.722,E2 35456.722} C_VEL
LIN {X 0,Y 751.957,Z 327.557,A -85,B 0,C 180,E1 35454.539,E2 35454.539} C_VEL
LIN {X 0,Y 751.038,Z 327.682,A -85,B 0,C 180,E1 35453.952,E2 35453.952} C_VEL
LIN {X 0,Y 744.514,Z 328.502,A -85,B 0,C 180,E1 35452.267,E2 35452.267} C_VEL
LIN {X 0,Y 744.026,Z 328.555,A -85,B 0,C 180,E1 35451.883,E2 35451.883} C_VEL
LIN {X 0,Y 743.967,Z 328.549,A -85,B 0,C 180,E1 35449.233,E2 35449.233} C_VEL
LIN {X 0,Y 743.989,Z 328.548,A -85,B 0,C 180,E1 35446.634,E2 35446.634} C_VEL
LIN {X 0,Y 744.006,Z 328.553,A -85,B 0,C 180,E1 35443.607,E2 35443.607} C_VEL
LIN {X 0,Y 743.967,Z 328.551,A -85,B 0,C 180,E1 35441.019,E2 35441.019} C_VEL
LIN {X 0,Y 743.996,Z 328.546,A -85,B 0,C 180,E1 35438.436,E2 35438.436} C_VEL
LIN {X 0,Y 743.995,Z 328.552,A -85,B 0,C 180,E1 35435.378,E2 35435.378} C_VEL
LIN {X 0,Y 743.967,Z 328.551,A -85,B 0,C 180,E1 35432.809,E2 35432.809} C_VEL
LIN {X 0,Y 744.012,Z 328.545,A -85,B 0,C 180,E1 35430.182,E2 35430.182} C_VEL
LIN {X 0,Y 743.992,Z 328.552,A -85,B 0,C 180,E1 35427.206,E2 35427.206} C_VEL
LIN {X 0,Y 743.968,Z 328.551,A -85,B 0,C 180,E1 35424.667,E2 35424.667} C_VEL
LIN {X 0,Y 744.023,Z 328.547,A -85,B 0,C 180,E1 35421.955,E2 35421.955} C_VEL
LIN {X 0,Y 743.988,Z 328.554,A -85,B 0,C 180,E1 35419.015,E2 35419.015} C_VEL
LIN {X 0,Y 743.968,Z 328.547,A -85,B 0,C 180,E1 35416.518,E2 35416.518} C_VEL
LIN {X 0,Y 744.029,Z 328.546,A -85,B 0,C 180,E1 35413.797,E2 35413.797} C_VEL
LIN {X 0,Y 743.985,Z 328.554,A -85,B 0,C 180,E1 35410.83,E2 35410.83} C_VEL
LIN {X 0,Y 743.971,Z 328.551,A -85,B 0,C 180,E1 35408.285,E2 35408.285} C_VEL
LIN {X 0,Y 744.033,Z 328.549,A -85,B 0,C 180,E1 35405.584,E2 35405.584} C_VEL
LIN {X 0,Y 744.036,Z 328.75,A -85,B 0,C 180,E1 35402.929,E2 35402.929} C_VEL
LIN {X 0,Y 745.502,Z 334.227,A -85,B 0,C 180,E1 35402.445,E2 35402.445} C_VEL
LIN {X 0,Y 745.558,Z 347.88,A -85,B 0,C 180,E1 35401.465,E2 35401.465} C_VEL
LIN {X 0,Y 746.434,Z 352.248,A -85,B 0,C 180,E1 35401.371,E2 35401.371} C_VEL
LIN {X 0,Y 746.09,Z 588.531,A -85,B 0,C 180,E1 35398.757,E2 35398.757} C_VEL
LIN {X 0,Y 745.863,Z 736.508,A -85,B 0,C 180,E1 35397.134,E2 35397.134} C_VEL
LIN {X 0,Y 745.725,Z 761.666,A -85,B 0,C 180,E1 35396.722,E2 35396.722} C_VEL
LIN {X 0,Y 745.624,Z 783.079,A -85,B 0,C 180,E1 35396.24,E2 35396.24} C_VEL
LIN {X 0,Y 745.497,Z 805.058,A -85,B 0,C 180,E1 35395.629,E2 35395.629} C_VEL
LIN {X 0,Y 745.324,Z 828.364,A -85,B 0,C 180,E1 35394.829,E2 35394.829} C_VEL
LIN {X 0,Y 745.183,Z 848.052,A -85,B 0,C 180,E1 35394.031,E2 35394.031} C_VEL
LIN {X 0,Y 744.976,Z 870.727,A -85,B 0,C 180,E1 35392.966,E2 35392.966} C_VEL
LIN {X 0,Y 744.819,Z 890.713,A -85,B 0,C 180,E1 35391.872,E2 35391.872} C_VEL
LIN {X 0,Y 744.633,Z 911.764,A -85,B 0,C 180,E1 35390.557,E2 35390.557} C_VEL
LIN {X 0,Y 744.494,Z 929.48,A -85,B 0,C 180,E1 35389.292,E2 35389.292} C_VEL
LIN {X 0,Y 744.334,Z 948.584,A -85,B 0,C 180,E1 35387.743,E2 35387.743} C_VEL
LIN {X 0,Y 744.247,Z 964.191,A -85,B 0,C 180,E1 35386.307,E2 35386.307} C_VEL
LIN {X 0,Y 744.133,Z 979.904,A -85,B 0,C 180,E1 35384.655,E2 35384.655} C_VEL
LIN {X 0,Y 744.062,Z 992.692,A -85,B 0,C 180,E1 35383.127,E2 35383.127} C_VEL
LIN {X 0,Y 744.001,Z 1005.783,A -85,B 0,C 180,E1 35381.316,E2 35381.316} C_VEL
LIN {X 0,Y 743.962,Z 1015.065,A -85,B 0,C 180,E1 35379.828,E2 35379.828} C_VEL
LIN {X 0,Y 743.94,Z 1024.68,A -85,B 0,C 180,E1 35378.035,E2 35378.035} C_VEL
LIN {X 0,Y 743.92,Z 1032.406,A -85,B 0,C 180,E1 35376.25,E2 35376.25} C_VEL
LIN {X 0,Y 743.907,Z 1038.397,A -85,B 0,C 180,E1 35374.548,E2 35374.548} C_VEL
LIN {X 0,Y 743.913,Z 1043.416,A -85,B 0,C 180,E1 35372.619,E2 35372.619} C_VEL
LIN {X 0,Y 743.915,Z 1046.286,A -85,B 0,C 180,E1 35371.001,E2 35371.001} C_VEL
LIN {X 0,Y 743.914,Z 1048.183,A -85,B 0,C 180,E1 35369.076,E2 35369.076} C_VEL
LIN {X 0,Y 743.893,Z 1048.318,A -85,B 0,C 180,E1 35367.304,E2 35367.304} C_VEL
LIN {X 0,Y 743.904,Z 1047.129,A -85,B 0,C 180,E1 35365.529,E2 35365.529} C_VEL
LIN {X 0,Y 743.913,Z 1044.199,A -85,B 0,C 180,E1 35363.672,E2 35363.672} C_VEL
LIN {X 0,Y 743.921,Z 1040.349,A -85,B 0,C 180,E1 35362.042,E2 35362.042} C_VEL
LIN {X 0,Y 743.911,Z 1034.101,A -85,B 0,C 180,E1 35360.093,E2 35360.093} C_VEL
LIN {X 0,Y 743.924,Z 1027.283,A -85,B 0,C 180,E1 35358.447,E2 35358.447} C_VEL
LIN {X 0,Y 743.953,Z 1019.092,A -85,B 0,C 180,E1 35356.792,E2 35356.792} C_VEL
LIN {X 0,Y 743.985,Z 1008.229,A -85,B 0,C 180,E1 35354.966,E2 35354.966} C_VEL
LIN {X 0,Y 744.044,Z 997.713,A -85,B 0,C 180,E1 35353.447,E2 35353.447} C_VEL
LIN {X 0,Y 744.124,Z 983.591,A -85,B 0,C 180,E1 35351.674,E2 35351.674} C_VEL
LIN {X 0,Y 744.185,Z 970.183,A -85,B 0,C 180,E1 35350.209,E2 35350.209} C_VEL
LIN {X 0,Y 744.322,Z 953.329,A -85,B 0,C 180,E1 35348.584,E2 35348.584} C_VEL
LIN {X 0,Y 744.428,Z 936.984,A -85,B 0,C 180,E1 35347.201,E2 35347.201} C_VEL
LIN {X 0,Y 744.595,Z 917.363,A -85,B 0,C 180,E1 35345.738,E2 35345.738} C_VEL
LIN {X 0,Y 744.726,Z 899.367,A -85,B 0,C 180,E1 35344.555,E2 35344.555} C_VEL
LIN {X 0,Y 744.936,Z 877.899,A -85,B 0,C 180,E1 35343.322,E2 35343.322} C_VEL
LIN {X 0,Y 745.08,Z 858.16,A -85,B 0,C 180,E1 35342.333,E2 35342.333} C_VEL
LIN {X 0,Y 745.301,Z 833.955,A -85,B 0,C 180,E1 35341.296,E2 35341.296} C_VEL
LIN {X 0,Y 745.412,Z 813.434,A -85,B 0,C 180,E1 35340.553,E2 35340.553} C_VEL
LIN {X 0,Y 745.617,Z 789.81,A -85,B 0,C 180,E1 35339.84,E2 35339.84} C_VEL
LIN {X 0,Y 745.707,Z 767.455,A -85,B 0,C 180,E1 35339.309,E2 35339.309} C_VEL
LIN {X 0,Y 745.812,Z 746.729,A -85,B 0,C 180,E1 35338.925,E2 35338.925} C_VEL
LIN {X 0,Y 745.905,Z 715.938,A -85,B 0,C 180,E1 35338.533,E2 35338.533} C_VEL
LIN {X 0,Y 746.291,Z 462.088,A -85,B 0,C 180,E1 35335.764,E2 35335.764} C_VEL
LIN {X 0,Y 746.261,Z 350.498,A -85,B 0,C 180,E1 35334.511,E2 35334.511} C_VEL
LIN {X 0,Y 745.481,Z 347.33,A -85,B 0,C 180,E1 35334.424,E2 35334.424} C_VEL
LIN {X 0,Y 745.285,Z 332.822,A -85,B 0,C 180,E1 35333.35,E2 35333.35} C_VEL
LIN {X 0,Y 744.016,Z 328.557,A -85,B 0,C 180,E1 35332.938,E2 35332.938} C_VEL
LIN {X 0,Y 743.986,Z 328.55,A -85,B 0,C 180,E1 35329.927,E2 35329.927} C_VEL
LIN {X 0,Y 743.969,Z 328.553,A -85,B 0,C 180,E1 35327.361,E2 35327.361} C_VEL
LIN {X 0,Y 744.036,Z 328.555,A -85,B 0,C 180,E1 35324.656,E2 35324.656} C_VEL
LIN {X 0,Y 743.977,Z 328.548,A -85,B 0,C 180,E1 35321.703,E2 35321.703} C_VEL
LIN {X 0,Y 743.971,Z 328.551,A -85,B 0,C 180,E1 35319.151,E2 35319.151} C_VEL
LIN {X 0,Y 744.038,Z 328.547,A -85,B 0,C 180,E1 35316.345,E2 35316.345} C_VEL
LIN {X 0,Y 743.975,Z 328.549,A -85,B 0,C 180,E1 35313.53,E2 35313.53} C_VEL
LIN {X 0,Y 743.972,Z 328.551,A -85,B 0,C 180,E1 35310.981,E2 35310.981} C_VEL
LIN {X 0,Y 744.039,Z 328.55,A -85,B 0,C 180,E1 35308.145,E2 35308.145} C_VEL
LIN {X 0,Y 743.973,Z 328.548,A -85,B 0,C 180,E1 35305.387,E2 35305.387} C_VEL
LIN {X 0,Y 743.972,Z 328.552,A -85,B 0,C 180,E1 35302.856,E2 35302.856} C_VEL
LIN {X 0,Y 744.038,Z 328.551,A -85,B 0,C 180,E1 35300.041,E2 35300.041} C_VEL
LIN {X 0,Y 743.971,Z 328.549,A -85,B 0,C 180,E1 35297.198,E2 35297.198} C_VEL
LIN {X 0,Y 743.972,Z 328.552,A -85,B 0,C 180,E1 35294.715,E2 35294.715} C_VEL
LIN {X 0,Y 744.039,Z 328.55,A -85,B 0,C 180,E1 35291.865,E2 35291.865} C_VEL
LIN {X 0,Y 743.97,Z 328.549,A -85,B 0,C 180,E1 35289.047,E2 35289.047} C_VEL
LIN {X 0,Y 743.971,Z 328.552,A -85,B 0,C 180,E1 35286.56,E2 35286.56} C_VEL
LIN {X 0,Y 744.038,Z 328.55,A -85,B 0,C 180,E1 35283.699,E2 35283.699} C_VEL
LIN {X 0,Y 743.971,Z 328.549,A -85,B 0,C 180,E1 35280.924,E2 35280.924} C_VEL
LIN {X 0,Y 743.969,Z 328.552,A -85,B 0,C 180,E1 35278.46,E2 35278.46} C_VEL
LIN {X 0,Y 744.039,Z 328.551,A -85,B 0,C 180,E1 35275.607,E2 35275.607} C_VEL
LIN {X 0,Y 743.971,Z 328.548,A -85,B 0,C 180,E1 35272.82,E2 35272.82} C_VEL
LIN {X 0,Y 743.968,Z 328.552,A -85,B 0,C 180,E1 35270.328,E2 35270.328} C_VEL
LIN {X 0,Y 744.038,Z 328.552,A -85,B 0,C 180,E1 35267.504,E2 35267.504} C_VEL
LIN {X 0,Y 743.973,Z 328.548,A -85,B 0,C 180,E1 35264.727,E2 35264.727} C_VEL
LIN {X 0,Y 743.966,Z 328.552,A -85,B 0,C 180,E1 35262.236,E2 35262.236} C_VEL
LIN {X 0,Y 744.037,Z 328.554,A -85,B 0,C 180,E1 35259.467,E2 35259.467} C_VEL
LIN {X 0,Y 743.976,Z 328.548,A -85,B 0,C 180,E1 35256.627,E2 35256.627} C_VEL
LIN {X 0,Y 743.963,Z 328.552,A -85,B 0,C 180,E1 35254.185,E2 35254.185} C_VEL
LIN {X 0,Y 744.021,Z 328.554,A -85,B 0,C 180,E1 35251.505,E2 35251.505} C_VEL
LIN {X 0,Y 743.981,Z 328.549,A -85,B 0,C 180,E1 35248.569,E2 35248.569} C_VEL
LIN {X 0,Y 743.963,Z 328.552,A -85,B 0,C 180,E1 35246.099,E2 35246.099} C_VEL
LIN {X 0,Y 744.006,Z 328.555,A -85,B 0,C 180,E1 35243.461,E2 35243.461} C_VEL
LIN {X 0,Y 743.987,Z 328.549,A -85,B 0,C 180,E1 35240.483,E2 35240.483} C_VEL
LIN {X 0,Y 743.963,Z 328.551,A -85,B 0,C 180,E1 35237.986,E2 35237.986} C_VEL
LIN {X 0,Y 743.993,Z 328.554,A -85,B 0,C 180,E1 35235.422,E2 35235.422} C_VEL
LIN {X 0,Y 743.986,Z 328.55,A -85,B 0,C 180,E1 35232.338,E2 35232.338} C_VEL
LIN {X 0,Y 743.962,Z 328.553,A -85,B 0,C 180,E1 35229.873,E2 35229.873} C_VEL
LIN {X 0,Y 743.98,Z 328.556,A -85,B 0,C 180,E1 35227.407,E2 35227.407} C_VEL
LIN {X 0,Y 744.045,Z 328.588,A -85,B 0,C 180,E1 35226.944,E2 35226.944} C_VEL
LIN {X 0,Y 745.78,Z 334.387,A -85,B 0,C 180,E1 35226.437,E2 35226.437} C_VEL
LIN {X 0,Y 745.596,Z 369.862,A -85,B 0,C 180,E1 35224.002,E2 35224.002} C_VEL
LIN {X 0,Y 745.658,Z 377.522,A -85,B 0,C 180,E1 35223.508,E2 35223.508} C_VEL
LIN {X 0,Y 746.472,Z 381.703,A -85,B 0,C 180,E1 35223.42,E2 35223.42} C_VEL
LIN {X 0,Y 746.062,Z 639.18,A -85,B 0,C 180,E1 35220.577,E2 35220.577} C_VEL
LIN {X 0,Y 745.862,Z 766.637,A -85,B 0,C 180,E1 35219.177,E2 35219.177} C_VEL
LIN {X 0,Y 745.723,Z 791.762,A -85,B 0,C 180,E1 35218.765,E2 35218.765} C_VEL
LIN {X 0,Y 745.624,Z 813.142,A -85,B 0,C 180,E1 35218.284,E2 35218.284} C_VEL
LIN {X 0,Y 745.497,Z 835.888,A -85,B 0,C 180,E1 35217.65,E2 35217.65} C_VEL
LIN {X 0,Y 745.319,Z 859.238,A -85,B 0,C 180,E1 35216.84,E2 35216.84} C_VEL
LIN {X 0,Y 745.177,Z 879.235,A -85,B 0,C 180,E1 35216.026,E2 35216.026} C_VEL
LIN {X 0,Y 744.961,Z 902.334,A -85,B 0,C 180,E1 35214.926,E2 35214.926} C_VEL
LIN {X 0,Y 744.818,Z 921.356,A -85,B 0,C 180,E1 35213.88,E2 35213.88} C_VEL
LIN {X 0,Y 744.619,Z 943.232,A -85,B 0,C 180,E1 35212.501,E2 35212.501} C_VEL
LIN {X 0,Y 744.488,Z 960.818,A -85,B 0,C 180,E1 35211.238,E2 35211.238} C_VEL
LIN {X 0,Y 744.337,Z 978.603,A -85,B 0,C 180,E1 35209.787,E2 35209.787} C_VEL
LIN {X 0,Y 744.244,Z 994.496,A -85,B 0,C 180,E1 35208.323,E2 35208.323} C_VEL
LIN {X 0,Y 744.133,Z 1009.8,A -85,B 0,C 180,E1 35206.711,E2 35206.711} C_VEL
LIN {X 0,Y 744.067,Z 1023.175,A -85,B 0,C 180,E1 35205.112,E2 35205.112} C_VEL
LIN {X 0,Y 744.007,Z 1035.899,A -85,B 0,C 180,E1 35203.343,E2 35203.343} C_VEL
LIN {X 0,Y 743.953,Z 1045.564,A -85,B 0,C 180,E1 35201.788,E2 35201.788} C_VEL
LIN {X 0,Y 743.922,Z 1055.47,A -85,B 0,C 180,E1 35199.907,E2 35199.907} C_VEL
LIN {X 0,Y 743.921,Z 1062.51,A -85,B 0,C 180,E1 35198.269,E2 35198.269} C_VEL
LIN {X 0,Y 743.897,Z 1068.506,A -85,B 0,C 180,E1 35196.56,E2 35196.56} C_VEL
LIN {X 0,Y 743.916,Z 1073.495,A -85,B 0,C 180,E1 35194.626,E2 35194.626} C_VEL
LIN {X 0,Y 743.912,Z 1076.459,A -85,B 0,C 180,E1 35192.928,E2 35192.928} C_VEL
LIN {X 0,Y 743.91,Z 1078.24,A -85,B 0,C 180,E1 35190.924,E2 35190.924} C_VEL
LIN {X 0,Y 743.894,Z 1078.306,A -85,B 0,C 180,E1 35189.307,E2 35189.307} C_VEL
LIN {X 0,Y 743.906,Z 1077.017,A -85,B 0,C 180,E1 35187.458,E2 35187.458} C_VEL
LIN {X 0,Y 743.901,Z 1073.971,A -85,B 0,C 180,E1 35185.606,E2 35185.606} C_VEL
LIN {X 0,Y 743.913,Z 1070.069,A -85,B 0,C 180,E1 35183.982,E2 35183.982} C_VEL
LIN {X 0,Y 743.916,Z 1063.726,A -85,B 0,C 180,E1 35182.042,E2 35182.042} C_VEL
LIN {X 0,Y 743.917,Z 1056.89,A -85,B 0,C 180,E1 35180.406,E2 35180.406} C_VEL
LIN {X 0,Y 743.973,Z 1047.87,A -85,B 0,C 180,E1 35178.605,E2 35178.605} C_VEL
LIN {X 0,Y 743.998,Z 1037.312,A -85,B 0,C 180,E1 35176.872,E2 35176.872} C_VEL
LIN {X 0,Y 744.045,Z 1026.214,A -85,B 0,C 180,E1 35175.286,E2 35175.286} C_VEL
LIN {X 0,Y 744.124,Z 1012.63,A -85,B 0,C 180,E1 35173.61,E2 35173.61} C_VEL
LIN {X 0,Y 744.184,Z 999.29,A -85,B 0,C 180,E1 35172.161,E2 35172.161} C_VEL
LIN {X 0,Y 744.331,Z 982.319,A -85,B 0,C 180,E1 35170.54,E2 35170.54} C_VEL
LIN {X 0,Y 744.429,Z 966.464,A -85,B 0,C 180,E1 35169.203,E2 35169.203} C_VEL
LIN {X 0,Y 744.599,Z 946.854,A -85,B 0,C 180,E1 35167.748,E2 35167.748} C_VEL
LIN {X 0,Y 744.739,Z 928.435,A -85,B 0,C 180,E1 35166.542,E2 35166.542} C_VEL
LIN {X 0,Y 744.94,Z 906.546,A -85,B 0,C 180,E1 35165.295,E2 35165.295} C_VEL
LIN {X 0,Y 745.09,Z 886.788,A -85,B 0,C 180,E1 35164.313,E2 35164.313} C_VEL
LIN {X 0,Y 745.305,Z 863.326,A -85,B 0,C 180,E1 35163.317,E2 35163.317} C_VEL
LIN {X 0,Y 745.413,Z 843.693,A -85,B 0,C 180,E1 35162.607,E2 35162.607} C_VEL
LIN {X 0,Y 745.617,Z 820.256,A -85,B 0,C 180,E1 35161.896,E2 35161.896} C_VEL
LIN {X 0,Y 745.705,Z 797.576,A -85,B 0,C 180,E1 35161.356,E2 35161.356} C_VEL
LIN {X 0,Y 745.809,Z 776.999,A -85,B 0,C 180,E1 35160.974,E2 35160.974} C_VEL
LIN {X 0,Y 745.904,Z 746.257,A -85,B 0,C 180,E1 35160.582,E2 35160.582} C_VEL
LIN {X 0,Y 746.271,Z 496.106,A -85,B 0,C 180,E1 35157.853,E2 35157.853} C_VEL
LIN {X 0,Y 746.29,Z 379.921,A -85,B 0,C 180,E1 35156.551,E2 35156.551} C_VEL
LIN {X 0,Y 745.547,Z 376.685,A -85,B 0,C 180,E1 35156.458,E2 35156.458} C_VEL
LIN {X 0,Y 745.733,Z 341.21,A -85,B 0,C 180,E1 35154.036,E2 35154.036} C_VEL
LIN {X 0,Y 745.691,Z 333.581,A -85,B 0,C 180,E1 35153.501,E2 35153.501} C_VEL
LIN {X 0,Y 744.039,Z 328.555,A -85,B 0,C 180,E1 35153.031,E2 35153.031} C_VEL
LIN {X 0,Y 743.965,Z 328.556,A -85,B 0,C 180,E1 35150.327,E2 35150.327} C_VEL
LIN {X 0,Y 743.969,Z 328.552,A -85,B 0,C 180,E1 35147.883,E2 35147.883} C_VEL
LIN {X 0,Y 744.04,Z 328.553,A -85,B 0,C 180,E1 35145.019,E2 35145.019} C_VEL
LIN {X 0,Y 743.968,Z 328.553,A -85,B 0,C 180,E1 35142.222,E2 35142.222} C_VEL
LIN {X 0,Y 743.968,Z 328.549,A -85,B 0,C 180,E1 35139.757,E2 35139.757} C_VEL
LIN {X 0,Y 744.037,Z 328.549,A -85,B 0,C 180,E1 35137.017,E2 35137.017} C_VEL
LIN {X 0,Y 743.973,Z 328.552,A -85,B 0,C 180,E1 35134.18,E2 35134.18} C_VEL
LIN {X 0,Y 743.964,Z 328.55,A -85,B 0,C 180,E1 35131.702,E2 35131.702} C_VEL
LIN {X 0,Y 744.041,Z 328.548,A -85,B 0,C 180,E1 35128.933,E2 35128.933} C_VEL
LIN {X 0,Y 743.976,Z 328.553,A -85,B 0,C 180,E1 35126.071,E2 35126.071} C_VEL
LIN {X 0,Y 743.966,Z 328.549,A -85,B 0,C 180,E1 35123.565,E2 35123.565} C_VEL
LIN {X 0,Y 744.033,Z 328.547,A -85,B 0,C 180,E1 35120.863,E2 35120.863} C_VEL
LIN {X 0,Y 743.976,Z 328.553,A -85,B 0,C 180,E1 35117.925,E2 35117.925} C_VEL
LIN {X 0,Y 743.966,Z 328.55,A -85,B 0,C 180,E1 35115.433,E2 35115.433} C_VEL
LIN {X 0,Y 744.039,Z 328.547,A -85,B 0,C 180,E1 35112.653,E2 35112.653} C_VEL
LIN {X 0,Y 743.973,Z 328.55,A -85,B 0,C 180,E1 35109.75,E2 35109.75} C_VEL
LIN {X 0,Y 743.968,Z 328.55,A -85,B 0,C 180,E1 35107.258,E2 35107.258} C_VEL
LIN {X 0,Y 744.038,Z 328.548,A -85,B 0,C 180,E1 35104.47,E2 35104.47} C_VEL
LIN {X 0,Y 743.975,Z 328.552,A -85,B 0,C 180,E1 35101.617,E2 35101.617} C_VEL
LIN {X 0,Y 743.97,Z 328.547,A -85,B 0,C 180,E1 35099.076,E2 35099.076} C_VEL
LIN {X 0,Y 744.039,Z 328.551,A -85,B 0,C 180,E1 35096.224,E2 35096.224} C_VEL
LIN {X 0,Y 743.973,Z 328.551,A -85,B 0,C 180,E1 35093.44,E2 35093.44} C_VEL
LIN {X 0,Y 744.026,Z 328.555,A -85,B 0,C 180,E1 35091.883,E2 35091.883} C_VEL
LIN {X 0,Y 742.975,Z 328.677,A -85,B 0,C 180,E1 35091.289,E2 35091.289} C_VEL
LIN {X 0,Y 736.559,Z 329.479,A -85,B 0,C 180,E1 35089.628,E2 35089.628} C_VEL
LIN {X 0,Y 736.028,Z 329.537,A -85,B 0,C 180,E1 35089.196,E2 35089.196} C_VEL
LIN {X 0,Y 736.058,Z 329.537,A -85,B 0,C 180,E1 35086.567,E2 35086.567} C_VEL
LIN {X 0,Y 736.055,Z 329.542,A -85,B 0,C 180,E1 35083.506,E2 35083.506} C_VEL
LIN {X 0,Y 736.029,Z 329.539,A -85,B 0,C 180,E1 35080.889,E2 35080.889} C_VEL
LIN {X 0,Y 736.093,Z 329.534,A -85,B 0,C 180,E1 35078.149,E2 35078.149} C_VEL
LIN {X 0,Y 736.045,Z 329.539,A -85,B 0,C 180,E1 35075.266,E2 35075.266} C_VEL
LIN {X 0,Y 736.032,Z 329.539,A -85,B 0,C 180,E1 35072.679,E2 35072.679} C_VEL
LIN {X 0,Y 736.101,Z 329.534,A -85,B 0,C 180,E1 35069.914,E2 35069.914} C_VEL
LIN {X 0,Y 736.037,Z 329.539,A -85,B 0,C 180,E1 35066.992,E2 35066.992} C_VEL
LIN {X 0,Y 736.036,Z 329.538,A -85,B 0,C 180,E1 35064.449,E2 35064.449} C_VEL
LIN {X 0,Y 736.1,Z 329.542,A -85,B 0,C 180,E1 35061.528,E2 35061.528} C_VEL
LIN {X 0,Y 736.035,Z 329.542,A -85,B 0,C 180,E1 35058.786,E2 35058.786} C_VEL
LIN {X 0,Y 736.041,Z 329.534,A -85,B 0,C 180,E1 35056.254,E2 35056.254} C_VEL
LIN {X 0,Y 736.095,Z 329.545,A -85,B 0,C 180,E1 35053.312,E2 35053.312} C_VEL
LIN {X 0,Y 736.033,Z 329.542,A -85,B 0,C 180,E1 35050.589,E2 35050.589} C_VEL
LIN {X 0,Y 736.053,Z 329.539,A -85,B 0,C 180,E1 35047.979,E2 35047.979} C_VEL
LIN {X 0,Y 736.074,Z 329.545,A -85,B 0,C 180,E1 35044.977,E2 35044.977} C_VEL
LIN {X 0,Y 736.135,Z 329.792,A -85,B 0,C 180,E1 35043.281,E2 35043.281} C_VEL
LIN {X 0,Y 738.337,Z 337.129,A -85,B 0,C 180,E1 35042.611,E2 35042.611} C_VEL
LIN {X 0,Y 738.378,Z 347.878,A -85,B 0,C 180,E1 35041.834,E2 35041.834} C_VEL
LIN {X 0,Y 739.744,Z 353.96,A -85,B 0,C 180,E1 35041.694,E2 35041.694} C_VEL
LIN {X 0,Y 739.21,Z 590.191,A -85,B 0,C 180,E1 35039.057,E2 35039.057} C_VEL
LIN {X 0,Y 738.867,Z 736.606,A -85,B 0,C 180,E1 35037.436,E2 35037.436} C_VEL
LIN {X 0,Y 738.668,Z 761.853,A -85,B 0,C 180,E1 35037.019,E2 35037.019} C_VEL
LIN {X 0,Y 738.513,Z 783.409,A -85,B 0,C 180,E1 35036.529,E2 35036.529} C_VEL
LIN {X 0,Y 738.317,Z 806.613,A -85,B 0,C 180,E1 35035.875,E2 35035.875} C_VEL
LIN {X 0,Y 738.049,Z 829.01,A -85,B 0,C 180,E1 35035.09,E2 35035.09} C_VEL
LIN {X 0,Y 737.831,Z 849.605,A -85,B 0,C 180,E1 35034.244,E2 35034.244} C_VEL
LIN {X 0,Y 737.513,Z 872.31,A -85,B 0,C 180,E1 35033.152,E2 35033.152} C_VEL
LIN {X 0,Y 737.286,Z 891.854,A -85,B 0,C 180,E1 35032.065,E2 35032.065} C_VEL
LIN {X 0,Y 736.995,Z 913.308,A -85,B 0,C 180,E1 35030.697,E2 35030.697} C_VEL
LIN {X 0,Y 736.792,Z 931.058,A -85,B 0,C 180,E1 35029.407,E2 35029.407} C_VEL
LIN {X 0,Y 736.554,Z 949.348,A -85,B 0,C 180,E1 35027.893,E2 35027.893} C_VEL
LIN {X 0,Y 736.416,Z 965.272,A -85,B 0,C 180,E1 35026.405,E2 35026.405} C_VEL
LIN {X 0,Y 736.243,Z 980.534,A -85,B 0,C 180,E1 35024.767,E2 35024.767} C_VEL
LIN {X 0,Y 736.145,Z 993.512,A -85,B 0,C 180,E1 35023.191,E2 35023.191} C_VEL
LIN {X 0,Y 736.049,Z 1005.935,A -85,B 0,C 180,E1 35021.44,E2 35021.44} C_VEL
LIN {X 0,Y 735.993,Z 1015.659,A -85,B 0,C 180,E1 35019.856,E2 35019.856} C_VEL
LIN {X 0,Y 735.94,Z 1025.705,A -85,B 0,C 180,E1 35017.918,E2 35017.918} C_VEL
LIN {X 0,Y 735.923,Z 1032.494,A -85,B 0,C 180,E1 35016.318,E2 35016.318} C_VEL
LIN {X 0,Y 735.911,Z 1038.47,A -85,B 0,C 180,E1 35014.598,E2 35014.598} C_VEL
LIN {X 0,Y 735.911,Z 1043.461,A -85,B 0,C 180,E1 35012.648,E2 35012.648} C_VEL
LIN {X 0,Y 735.914,Z 1046.318,A -85,B 0,C 180,E1 35011.012,E2 35011.012} C_VEL
LIN {X 0,Y 735.914,Z 1048.189,A -85,B 0,C 180,E1 35009.066,E2 35009.066} C_VEL
LIN {X 0,Y 735.892,Z 1048.334,A -85,B 0,C 180,E1 35007.352,E2 35007.352} C_VEL
LIN {X 0,Y 735.912,Z 1047.245,A -85,B 0,C 180,E1 35005.636,E2 35005.636} C_VEL
LIN {X 0,Y 735.913,Z 1044.313,A -85,B 0,C 180,E1 35003.681,E2 35003.681} C_VEL
LIN {X 0,Y 735.923,Z 1040.497,A -85,B 0,C 180,E1 35002.034,E2 35002.034} C_VEL
LIN {X 0,Y 735.915,Z 1034.623,A -85,B 0,C 180,E1 35000.143,E2 35000.143} C_VEL
LIN {X 0,Y 735.935,Z 1027.538,A -85,B 0,C 180,E1 34998.4,E2 34998.4} C_VEL
LIN {X 0,Y 735.973,Z 1019.795,A -85,B 0,C 180,E1 34996.806,E2 34996.806} C_VEL
LIN {X 0,Y 736.032,Z 1008.602,A -85,B 0,C 180,E1 34994.881,E2 34994.881} C_VEL
LIN {X 0,Y 736.11,Z 998.128,A -85,B 0,C 180,E1 34993.345,E2 34993.345} C_VEL
LIN {X 0,Y 736.227,Z 984.804,A -85,B 0,C 180,E1 34991.634,E2 34991.634} C_VEL
LIN {X 0,Y 736.328,Z 970.74,A -85,B 0,C 180,E1 34990.072,E2 34990.072} C_VEL
LIN {X 0,Y 736.53,Z 954.755,A -85,B 0,C 180,E1 34988.497,E2 34988.497} C_VEL
LIN {X 0,Y 736.69,Z 938.221,A -85,B 0,C 180,E1 34987.074,E2 34987.074} C_VEL
LIN {X 0,Y 736.94,Z 919.455,A -85,B 0,C 180,E1 34985.64,E2 34985.64} C_VEL
LIN {X 0,Y 737.138,Z 901.371,A -85,B 0,C 180,E1 34984.428,E2 34984.428} C_VEL
LIN {X 0,Y 737.451,Z 880.688,A -85,B 0,C 180,E1 34983.203,E2 34983.203} C_VEL
LIN {X 0,Y 737.672,Z 860.35,A -85,B 0,C 180,E1 34982.163,E2 34982.163} C_VEL
LIN {X 0,Y 737.971,Z 838.881,A -85,B 0,C 180,E1 34981.205,E2 34981.205} C_VEL
LIN {X 0,Y 738.184,Z 815.929,A -85,B 0,C 180,E1 34980.347,E2 34980.347} C_VEL
LIN {X 0,Y 738.404,Z 794.836,A -85,B 0,C 180,E1 34979.685,E2 34979.685} C_VEL
LIN {X 0,Y 738.632,Z 769.892,A -85,B 0,C 180,E1 34979.061,E2 34979.061} C_VEL
LIN {X 0,Y 738.783,Z 749.231,A -85,B 0,C 180,E1 34978.665,E2 34978.665} C_VEL
LIN {X 0,Y 738.911,Z 725.248,A -85,B 0,C 180,E1 34978.329,E2 34978.329} C_VEL
LIN {X 0,Y 739.488,Z 471.878,A -85,B 0,C 180,E1 34975.542,E2 34975.542} C_VEL
LIN {X 0,Y 739.552,Z 352.325,A -85,B 0,C 180,E1 34974.188,E2 34974.188} C_VEL
LIN {X 0,Y 738.297,Z 347.255,A -85,B 0,C 180,E1 34974.049,E2 34974.049} C_VEL
LIN {X 0,Y 738.215,Z 336.227,A -85,B 0,C 180,E1 34973.225,E2 34973.225} C_VEL
LIN {X 0,Y 736.1,Z 329.543,A -85,B 0,C 180,E1 34972.589,E2 34972.589} C_VEL
LIN {X 0,Y 736.035,Z 329.541,A -85,B 0,C 180,E1 34969.771,E2 34969.771} C_VEL
LIN {X 0,Y 736.039,Z 329.544,A -85,B 0,C 180,E1 34967.187,E2 34967.187} C_VEL
LIN {X 0,Y 736.099,Z 329.536,A -85,B 0,C 180,E1 34964.283,E2 34964.283} C_VEL
LIN {X 0,Y 736.029,Z 329.538,A -85,B 0,C 180,E1 34961.525,E2 34961.525} C_VEL
LIN {X 0,Y 736.044,Z 329.541,A -85,B 0,C 180,E1 34958.974,E2 34958.974} C_VEL
LIN {X 0,Y 736.076,Z 329.53,A -85,B 0,C 180,E1 34955.942,E2 34955.942} C_VEL
LIN {X 0,Y 736.028,Z 329.54,A -85,B 0,C 180,E1 34953.287,E2 34953.287} C_VEL
LIN {X 0,Y 736.068,Z 329.542,A -85,B 0,C 180,E1 34950.625,E2 34950.625} C_VEL
LIN {X 0,Y 736.05,Z 329.538,A -85,B 0,C 180,E1 34947.596,E2 34947.596} C_VEL
LIN {X 0,Y 736.027,Z 329.539,A -85,B 0,C 180,E1 34945.026,E2 34945.026} C_VEL
LIN {X 0,Y 736.094,Z 329.543,A -85,B 0,C 180,E1 34942.271,E2 34942.271} C_VEL
LIN {X 0,Y 736.041,Z 329.538,A -85,B 0,C 180,E1 34939.358,E2 34939.358} C_VEL
LIN {X 0,Y 736.03,Z 329.54,A -85,B 0,C 180,E1 34936.82,E2 34936.82} C_VEL
LIN {X 0,Y 736.1,Z 329.54,A -85,B 0,C 180,E1 34933.992,E2 34933.992} C_VEL
LIN {X 0,Y 736.033,Z 329.538,A -85,B 0,C 180,E1 34931.122,E2 34931.122} C_VEL
LIN {X 0,Y 736.033,Z 329.541,A -85,B 0,C 180,E1 34928.594,E2 34928.594} C_VEL
LIN {X 0,Y 736.1,Z 329.538,A -85,B 0,C 180,E1 34925.769,E2 34925.769} C_VEL
LIN {X 0,Y 736.032,Z 329.539,A -85,B 0,C 180,E1 34922.959,E2 34922.959} C_VEL
LIN {X 0,Y 736.033,Z 329.54,A -85,B 0,C 180,E1 34920.467,E2 34920.467} C_VEL
LIN {X 0,Y 736.099,Z 329.538,A -85,B 0,C 180,E1 34917.664,E2 34917.664} C_VEL
LIN {X 0,Y 736.033,Z 329.539,A -85,B 0,C 180,E1 34914.856,E2 34914.856} C_VEL
LIN {X 0,Y 736.03,Z 329.539,A -85,B 0,C 180,E1 34912.349,E2 34912.349} C_VEL
LIN {X 0,Y 736.099,Z 329.537,A -85,B 0,C 180,E1 34909.512,E2 34909.512} C_VEL
LIN {X 0,Y 736.033,Z 329.539,A -85,B 0,C 180,E1 34906.727,E2 34906.727} C_VEL
LIN {X 0,Y 736.029,Z 329.539,A -85,B 0,C 180,E1 34904.235,E2 34904.235} C_VEL
LIN {X 0,Y 736.1,Z 329.537,A -85,B 0,C 180,E1 34901.384,E2 34901.384} C_VEL
LIN {X 0,Y 736.029,Z 329.539,A -85,B 0,C 180,E1 34898.523,E2 34898.523} C_VEL
LIN {X 0,Y 736.032,Z 329.539,A -85,B 0,C 180,E1 34896.034,E2 34896.034} C_VEL
LIN {X 0,Y 736.101,Z 329.538,A -85,B 0,C 180,E1 34893.182,E2 34893.182} C_VEL
LIN {X 0,Y 736.029,Z 329.539,A -85,B 0,C 180,E1 34890.393,E2 34890.393} C_VEL
LIN {X 0,Y 736.03,Z 329.542,A -85,B 0,C 180,E1 34887.915,E2 34887.915} C_VEL
LIN {X 0,Y 736.099,Z 329.541,A -85,B 0,C 180,E1 34885.119,E2 34885.119} C_VEL
LIN {X 0,Y 736.032,Z 329.539,A -85,B 0,C 180,E1 34882.315,E2 34882.315} C_VEL
LIN {X 0,Y 736.028,Z 329.542,A -85,B 0,C 180,E1 34879.813,E2 34879.813} C_VEL
LIN {X 0,Y 736.098,Z 329.542,A -85,B 0,C 180,E1 34877.007,E2 34877.007} C_VEL
LIN {X 0,Y 736.032,Z 329.54,A -85,B 0,C 180,E1 34874.169,E2 34874.169} C_VEL
LIN {X 0,Y 736.031,Z 329.543,A -85,B 0,C 180,E1 34871.629,E2 34871.629} C_VEL
LIN {X 0,Y 736.101,Z 329.543,A -85,B 0,C 180,E1 34868.767,E2 34868.767} C_VEL
LIN {X 0,Y 736.058,Z 329.629,A -85,B 0,C 180,E1 34867.339,E2 34867.339} C_VEL
LIN {X 0,Y 738.755,Z 337.51,A -85,B 0,C 180,E1 34866.619,E2 34866.619} C_VEL
LIN {X 0,Y 738.447,Z 373.273,A -85,B 0,C 180,E1 34864.142,E2 34864.142} C_VEL
LIN {X 0,Y 738.5,Z 377.442,A -85,B 0,C 180,E1 34863.878,E2 34863.878} C_VEL
LIN {X 0,Y 739.785,Z 383.425,A -85,B 0,C 180,E1 34863.743,E2 34863.743} C_VEL
LIN {X 0,Y 739.163,Z 641.852,A -85,B 0,C 180,E1 34860.864,E2 34860.864} C_VEL
LIN {X 0,Y 738.866,Z 766.745,A -85,B 0,C 180,E1 34859.479,E2 34859.479} C_VEL
LIN {X 0,Y 738.666,Z 792.02,A -85,B 0,C 180,E1 34859.061,E2 34859.061} C_VEL
LIN {X 0,Y 738.512,Z 813.469,A -85,B 0,C 180,E1 34858.573,E2 34858.573} C_VEL
LIN {X 0,Y 738.321,Z 836.62,A -85,B 0,C 180,E1 34857.92,E2 34857.92} C_VEL
LIN {X 0,Y 738.045,Z 859.542,A -85,B 0,C 180,E1 34857.115,E2 34857.115} C_VEL
LIN {X 0,Y 737.827,Z 880.233,A -85,B 0,C 180,E1 34856.261,E2 34856.261} C_VEL
LIN {X 0,Y 737.503,Z 903.14,A -85,B 0,C 180,E1 34855.153,E2 34855.153} C_VEL
